Staubli VAL3: Robotscan.dtx

bool bSignal = true
bool bTxt1
bool bTxt2
bool bTxt3
bool btrig
public dio fout = {link=fOut0}
public frame FrmDraw = {x=1000, y=-100, fatherId=world[0]}
mdesc mNomSpeed
num l_nInit = 1500
num nNumTotal = 5031
num nNumrecord = 220
public num nTranC[6]
  [0] = 978.504226
  [1] = -109.919125
  [2] = 104.826018
  [3] = -0.09799
  [4] = 179.816018
  [5] = 56.0978696
num nTxtTotal = 11
num n_sTxt = 3
num ndelay = 16.304
public num nnnn = 2
num ntime = 2423.6
pointRx pfrmCad[1500]
  [0] = {x=-21.496, y=-9.92, z=104.826, rx=179.902, ry=0.184, rz=-123.901, fatherId=FrmDraw[0]}
  [1] = {x=-21.406, y=-9.571, z=104.833, rx=179.906, ry=0.177, rz=-124.352, fatherId=FrmDraw[0]}
  [2] = {x=-21.327, y=-9.235, z=104.84, rx=179.91, ry=0.172, rz=-124.769, fatherId=FrmDraw[0]}
  [3] = {x=-21.269, y=-8.967, z=104.845, rx=179.913, ry=0.168, rz=-125.087, fatherId=FrmDraw[0]}
  [4] = {x=-21.197, y=-8.609, z=104.852, rx=179.915, ry=0.164, rz=-125.501, fatherId=FrmDraw[0]}
  [5] = {x=-21.125, y=-8.284, z=104.858, rx=179.919, ry=0.159, rz=-125.914, fatherId=FrmDraw[0]}
  [6] = {x=-21.063, y=-8.029, z=104.863, rx=179.922, ry=0.154, rz=-126.277, fatherId=FrmDraw[0]}
  [7] = {x=-20.979, y=-7.711, z=104.871, rx=179.927, ry=0.146, rz=-126.778, fatherId=FrmDraw[0]}
  [8] = {x=-20.888, y=-7.402, z=104.879, rx=179.933, ry=0.136, rz=-127.324, fatherId=FrmDraw[0]}
  [9] = {x=-20.796, y=-7.121, z=104.886, rx=179.939, ry=0.125, rz=-127.88, fatherId=FrmDraw[0]}
  [10] = {x=-20.693, y=-6.864, z=104.895, rx=179.946, ry=0.112, rz=-128.514, fatherId=FrmDraw[0]}
  [11] = {x=-20.565, y=-6.611, z=104.905, rx=179.956, ry=0.094, rz=-129.312, fatherId=FrmDraw[0]}
  [12] = {x=-20.433, y=-6.398, z=104.914, rx=179.965, ry=0.076, rz=-130.171, fatherId=FrmDraw[0]}
  [13] = {x=-20.305, y=-6.222, z=104.923, rx=179.973, ry=0.059, rz=-131.051, fatherId=FrmDraw[0]}
  [14] = {x=-20.156, y=-6.043, z=104.933, rx=179.981, ry=0.042, rz=-132.148, fatherId=FrmDraw[0]}
  [15] = {x=-20.038, y=-5.901, z=104.94, rx=179.986, ry=0.032, rz=-133.098, fatherId=FrmDraw[0]}
  [16] = {x=-19.899, y=-5.734, z=104.948, rx=179.99, ry=0.023, rz=-134.309, fatherId=FrmDraw[0]}
  [17] = {x=-19.764, y=-5.576, z=104.955, rx=179.993, ry=0.017, rz=-135.558, fatherId=FrmDraw[0]}
  [18] = {x=-19.634, y=-5.431, z=104.961, rx=179.995, ry=0.013, rz=-136.824, fatherId=FrmDraw[0]}
  [19] = {x=-19.514, y=-5.306, z=104.967, rx=179.997, ry=0.008, rz=-138.02, fatherId=FrmDraw[0]}
  [20] = {x=-19.402, y=-5.193, z=104.973, rx=179.998, ry=0.005, rz=-139.156, fatherId=FrmDraw[0]}
  [21] = {x=-19.268, y=-5.059, z=104.979, rx=-180, rz=-140.558, fatherId=FrmDraw[0]}
  [22] = {x=-19.155, y=-4.95, z=104.985, rx=-179.999, ry=-0.004, rz=-141.768, fatherId=FrmDraw[0]}
  [23] = {x=-19.052, y=-4.852, z=104.99, rx=-179.997, ry=-0.008, rz=-142.893, fatherId=FrmDraw[0]}
  [24] = {x=-18.935, y=-4.744, z=104.995, rx=-179.996, ry=-0.013, rz=-144.181, fatherId=FrmDraw[0]}
  [25] = {x=-18.824, y=-4.636, z=105.001, rx=-179.995, ry=-0.017, rz=-145.451, fatherId=FrmDraw[0]}
  [26] = {x=-18.703, y=-4.509, z=105.006, rx=-179.994, ry=-0.021, rz=-146.89, fatherId=FrmDraw[0]}
  [27] = {x=-18.592, y=-4.383, z=105.011, rx=-179.993, ry=-0.023, rz=-148.26, fatherId=FrmDraw[0]}
  [28] = {x=-18.492, y=-4.26, z=105.016, rx=-179.993, ry=-0.024, rz=-149.572, fatherId=FrmDraw[0]}
  [29] = {x=-18.401, y=-4.137, z=105.02, rx=-179.994, ry=-0.023, rz=-150.833, fatherId=FrmDraw[0]}
  [30] = {x=-18.318, y=-4.016, z=105.023, rx=-179.995, ry=-0.022, rz=-152.05, fatherId=FrmDraw[0]}
  [31] = {x=-18.223, y=-3.864, z=105.027, rx=-179.996, ry=-0.017, rz=-153.555, fatherId=FrmDraw[0]}
  [32] = {x=-18.157, y=-3.747, z=105.029, rx=-179.997, ry=-0.012, rz=-154.683, fatherId=FrmDraw[0]}
  [33] = {x=-18.097, y=-3.632, z=105.031, rx=-179.999, ry=-0.006, rz=-155.782, fatherId=FrmDraw[0]}
  [34] = {x=-18.044, y=-3.519, z=105.032, rx=180, ry=0.001, rz=-156.854, fatherId=FrmDraw[0]}
  [35] = {x=-17.996, y=-3.408, z=105.033, rx=179.998, ry=0.01, rz=-157.905, fatherId=FrmDraw[0]}
  [36] = {x=-17.952, y=-3.3, z=105.034, rx=179.996, ry=0.019, rz=-158.942, fatherId=FrmDraw[0]}
  [37] = {x=-17.893, y=-3.145, z=105.035, rx=179.994, ry=0.034, rz=-160.472, fatherId=FrmDraw[0]}
  [38] = {x=-17.842, y=-2.998, z=105.035, rx=179.992, ry=0.05, rz=-161.989, fatherId=FrmDraw[0]}
  [39] = {x=-17.798, y=-2.858, z=105.034, rx=179.99, ry=0.068, rz=-163.483, fatherId=FrmDraw[0]}
  [40] = {x=-17.759, y=-2.726, z=105.033, rx=179.989, ry=0.087, rz=-164.962, fatherId=FrmDraw[0]}
  [41] = {x=-17.726, y=-2.601, z=105.032, rx=179.987, ry=0.106, rz=-166.428, fatherId=FrmDraw[0]}
  [42] = {x=-17.699, y=-2.483, z=105.03, rx=179.987, ry=0.127, rz=-167.883, fatherId=FrmDraw[0]}
  [43] = {x=-17.676, y=-2.372, z=105.028, rx=179.986, ry=0.148, rz=-169.329, fatherId=FrmDraw[0]}
  [44] = {x=-17.657, y=-2.266, z=105.026, rx=179.986, ry=0.17, rz=-170.767, fatherId=FrmDraw[0]}
  [45] = {x=-17.643, y=-2.167, z=105.023, rx=179.987, ry=0.193, rz=-172.197, fatherId=FrmDraw[0]}
  [46] = {x=-17.635, y=-2.07, z=105.02, rx=179.988, ry=0.217, rz=-173.604, fatherId=FrmDraw[0]}
  [47] = {x=-17.631, y=-1.974, z=105.016, rx=179.989, ry=0.242, rz=-174.986, fatherId=FrmDraw[0]}
  [48] = {x=-17.632, y=-1.879, z=105.012, rx=179.991, ry=0.268, rz=-176.347, fatherId=FrmDraw[0]}
  [49] = {x=-17.636, y=-1.787, z=105.008, rx=179.994, ry=0.293, rz=-177.689, fatherId=FrmDraw[0]}
  [50] = {x=-17.643, y=-1.696, z=105.004, rx=179.997, ry=0.319, rz=-179.015, fatherId=FrmDraw[0]}
  [51] = {x=-17.654, y=-1.579, z=104.998, rx=-179.998, ry=0.353, rz=179.235, fatherId=FrmDraw[0]}
  [52] = {x=-17.666, y=-1.469, z=104.993, rx=-179.992, ry=0.384, rz=177.491, fatherId=FrmDraw[0]}
  [53] = {x=-17.679, y=-1.366, z=104.987, rx=-179.985, ry=0.414, rz=175.749, fatherId=FrmDraw[0]}
  [54] = {x=-17.691, y=-1.271, z=104.982, rx=-179.977, ry=0.442, rz=174.006, fatherId=FrmDraw[0]}
  [55] = {x=-17.704, y=-1.183, z=104.977, rx=-179.968, ry=0.469, rz=172.258, fatherId=FrmDraw[0]}
  [56] = {x=-17.721, y=-1.092, z=104.972, rx=-179.959, ry=0.496, rz=170.546, fatherId=FrmDraw[0]}
  [57] = {x=-17.744, y=-0.993, z=104.966, rx=-179.949, ry=0.523, rz=168.902, fatherId=FrmDraw[0]}
  [58] = {x=-17.774, y=-0.886, z=104.96, rx=-179.939, ry=0.552, rz=167.322, fatherId=FrmDraw[0]}
  [59] = {x=-17.809, y=-0.77, z=104.954, rx=-179.928, ry=0.582, rz=165.802, fatherId=FrmDraw[0]}
  [60] = {x=-17.851, y=-0.646, z=104.947, rx=-179.916, ry=0.612, rz=164.339, fatherId=FrmDraw[0]}
  [61] = {x=-17.898, y=-0.515, z=104.94, rx=-179.903, ry=0.644, rz=162.93, fatherId=FrmDraw[0]}
  [62] = {x=-17.951, y=-0.376, z=104.932, rx=-179.89, ry=0.676, rz=161.572, fatherId=FrmDraw[0]}
  [63] = {x=-18.009, y=-0.231, z=104.925, rx=-179.877, ry=0.708, rz=160.261, fatherId=FrmDraw[0]}
  [64] = {x=-18.071, y=-0.079, z=104.917, rx=-179.863, ry=0.741, rz=158.995, fatherId=FrmDraw[0]}
  [65] = {x=-18.137, y=0.079, z=104.908, rx=-179.848, ry=0.775, rz=157.77, fatherId=FrmDraw[0]}
  [66] = {x=-18.207, y=0.239, z=104.9, rx=-179.833, ry=0.807, rz=156.562, fatherId=FrmDraw[0]}
  [67] = {x=-18.277, y=0.395, z=104.892, rx=-179.817, ry=0.839, rz=155.349, fatherId=FrmDraw[0]}
  [68] = {x=-18.35, y=0.548, z=104.885, rx=-179.8, ry=0.869, rz=154.132, fatherId=FrmDraw[0]}
  [69] = {x=-18.426, y=0.698, z=104.877, rx=-179.784, ry=0.898, rz=152.908, fatherId=FrmDraw[0]}
  [70] = {x=-18.504, y=0.844, z=104.869, rx=-179.766, ry=0.927, rz=151.676, fatherId=FrmDraw[0]}
  [71] = {x=-18.584, y=0.987, z=104.861, rx=-179.748, ry=0.955, rz=150.435, fatherId=FrmDraw[0]}
  [72] = {x=-18.668, y=1.126, z=104.854, rx=-179.729, ry=0.983, rz=149.184, fatherId=FrmDraw[0]}
  [73] = {x=-18.756, y=1.261, z=104.846, rx=-179.71, ry=1.01, rz=147.922, fatherId=FrmDraw[0]}
  [74] = {x=-18.847, y=1.391, z=104.838, rx=-179.689, ry=1.037, rz=146.647, fatherId=FrmDraw[0]}
  [75] = {x=-18.943, y=1.517, z=104.83, rx=-179.668, ry=1.064, rz=145.357, fatherId=FrmDraw[0]}
  [76] = {x=-19.043, y=1.64, z=104.821, rx=-179.646, ry=1.092, rz=144.066, fatherId=FrmDraw[0]}
  [77] = {x=-19.149, y=1.767, z=104.812, rx=-179.623, ry=1.121, rz=142.804, fatherId=FrmDraw[0]}
  [78] = {x=-19.258, y=1.9, z=104.803, rx=-179.599, ry=1.151, rz=141.57, fatherId=FrmDraw[0]}
  [79] = {x=-19.315, y=1.968, z=104.799, rx=-179.587, ry=1.166, rz=140.964, fatherId=FrmDraw[0]}
  [80] = {x=-19.401, y=2.072, z=104.792, rx=-179.568, ry=1.19, rz=140.069, fatherId=FrmDraw[0]}
  [81] = {x=-19.518, y=2.217, z=104.782, rx=-179.542, ry=1.221, rz=138.9, fatherId=FrmDraw[0]}
  [82] = {x=-19.638, y=2.368, z=104.772, rx=-179.516, ry=1.252, rz=137.76, fatherId=FrmDraw[0]}
  [83] = {x=-19.759, y=2.525, z=104.763, rx=-179.49, ry=1.282, rz=136.648, fatherId=FrmDraw[0]}
  [84] = {x=-19.88, y=2.688, z=104.754, rx=-179.464, ry=1.312, rz=135.564, fatherId=FrmDraw[0]}
  [85] = {x=-20.001, y=2.86, z=104.745, rx=-179.438, ry=1.34, rz=134.508, fatherId=FrmDraw[0]}
  [86] = {x=-20.122, y=3.039, z=104.736, rx=-179.412, ry=1.367, rz=133.478, fatherId=FrmDraw[0]}
  [87] = {x=-20.24, y=3.225, z=104.728, rx=-179.387, ry=1.391, rz=132.471, fatherId=FrmDraw[0]}
  [88] = {x=-20.358, y=3.418, z=104.721, rx=-179.363, ry=1.413, rz=131.482, fatherId=FrmDraw[0]}
  [89] = {x=-20.475, y=3.617, z=104.714, rx=-179.339, ry=1.434, rz=130.511, fatherId=FrmDraw[0]}
  [90] = {x=-20.592, y=3.823, z=104.707, rx=-179.316, ry=1.453, rz=129.559, fatherId=FrmDraw[0]}
  [91] = {x=-20.71, y=4.035, z=104.701, rx=-179.293, ry=1.471, rz=128.624, fatherId=FrmDraw[0]}
  [92] = {x=-20.823, y=4.242, z=104.695, rx=-179.271, ry=1.487, rz=127.752, fatherId=FrmDraw[0]}
  [93] = {x=-20.943, y=4.465, z=104.689, rx=-179.248, ry=1.504, rz=126.851, fatherId=FrmDraw[0]}
  [94] = {x=-21.066, y=4.694, z=104.683, rx=-179.224, ry=1.521, rz=125.967, fatherId=FrmDraw[0]}
  [95] = {x=-21.192, y=4.928, z=104.677, rx=-179.201, ry=1.538, rz=125.099, fatherId=FrmDraw[0]}
  [96] = {x=-21.321, y=5.168, z=104.67, rx=-179.177, ry=1.556, rz=124.249, fatherId=FrmDraw[0]}
  [97] = {x=-21.453, y=5.415, z=104.664, rx=-179.153, ry=1.575, rz=123.427, fatherId=FrmDraw[0]}
  [98] = {x=-21.587, y=5.671, z=104.658, rx=-179.128, ry=1.594, rz=122.636, fatherId=FrmDraw[0]}
  [99] = {x=-21.722, y=5.937, z=104.652, rx=-179.103, ry=1.615, rz=121.878, fatherId=FrmDraw[0]}
  [100] = {x=-21.857, y=6.213, z=104.646, rx=-179.078, ry=1.635, rz=121.155, fatherId=FrmDraw[0]}
  [101] = {x=-21.99, y=6.5, z=104.64, rx=-179.053, ry=1.655, rz=120.468, fatherId=FrmDraw[0]}
  [102] = {x=-22.118, y=6.791, z=104.635, rx=-179.03, ry=1.674, rz=119.831, fatherId=FrmDraw[0]}
  [103] = {x=-22.226, y=7.051, z=104.631, rx=-179.011, ry=1.69, rz=119.312, fatherId=FrmDraw[0]}
  [104] = {x=-22.313, y=7.274, z=104.628, rx=-178.995, ry=1.702, rz=118.9, fatherId=FrmDraw[0]}
  [105] = {x=-22.431, y=7.598, z=104.624, rx=-178.975, ry=1.718, rz=118.352, fatherId=FrmDraw[0]}
  [106] = {x=-22.528, y=7.887, z=104.622, rx=-178.958, ry=1.731, rz=117.91, fatherId=FrmDraw[0]}
  [107] = {x=-22.602, y=8.124, z=104.62, rx=-178.946, ry=1.74, rz=117.572, fatherId=FrmDraw[0]}
  [108] = {x=-22.692, y=8.429, z=104.618, rx=-178.931, ry=1.75, rz=117.171, fatherId=FrmDraw[0]}
  [109] = {x=-22.762, y=8.68, z=104.617, rx=-178.92, ry=1.757, rz=116.866, fatherId=FrmDraw[0]}
  [110] = {x=-22.845, y=9.001, z=104.617, rx=-178.908, ry=1.765, rz=116.506, fatherId=FrmDraw[0]}
  [111] = {x=-22.909, y=9.265, z=104.616, rx=-178.898, ry=1.772, rz=116.235, fatherId=FrmDraw[0]}
  [112] = {x=-22.985, y=9.602, z=104.616, rx=-178.887, ry=1.779, rz=115.918, fatherId=FrmDraw[0]}
  [113] = {x=-23.044, y=9.878, z=104.616, rx=-178.878, ry=1.784, rz=115.682, fatherId=FrmDraw[0]}
  [114] = {x=-23.114, y=10.232, z=104.616, rx=-178.868, ry=1.791, rz=115.409, fatherId=FrmDraw[0]}
  [115] = {x=-23.168, y=10.52, z=104.617, rx=-178.86, ry=1.797, rz=115.209, fatherId=FrmDraw[0]}
  [116] = {x=-23.231, y=10.889, z=104.617, rx=-178.85, ry=1.804, rz=114.981, fatherId=FrmDraw[0]}
  [117] = {x=-23.28, y=11.188, z=104.618, rx=-178.843, ry=1.809, rz=114.813, fatherId=FrmDraw[0]}
  [118] = {x=-23.341, y=11.564, z=104.619, rx=-178.834, ry=1.816, rz=114.603, fatherId=FrmDraw[0]}
  [119] = {x=-23.391, y=11.865, z=104.62, rx=-178.827, ry=1.821, rz=114.433, fatherId=FrmDraw[0]}
  [120] = {x=-23.455, y=12.243, z=104.621, rx=-178.819, ry=1.827, rz=114.218, fatherId=FrmDraw[0]}
  [121] = {x=-23.507, y=12.545, z=104.623, rx=-178.812, ry=1.831, rz=114.045, fatherId=FrmDraw[0]}
  [122] = {x=-23.573, y=12.924, z=104.624, rx=-178.804, ry=1.836, rz=113.827, fatherId=FrmDraw[0]}
  [123] = {x=-23.626, y=13.227, z=104.625, rx=-178.797, ry=1.84, rz=113.651, fatherId=FrmDraw[0]}
  [124] = {x=-23.695, y=13.607, z=104.627, rx=-178.789, ry=1.844, rz=113.428, fatherId=FrmDraw[0]}
  [125] = {x=-23.751, y=13.912, z=104.628, rx=-178.783, ry=1.847, rz=113.248, fatherId=FrmDraw[0]}
  [126] = {x=-23.823, y=14.293, z=104.63, rx=-178.775, ry=1.851, rz=113.022, fatherId=FrmDraw[0]}
  [127] = {x=-23.882, y=14.598, z=104.632, rx=-178.769, ry=1.854, rz=112.839, fatherId=FrmDraw[0]}
  [128] = {x=-23.957, y=14.981, z=104.634, rx=-178.761, ry=1.858, rz=112.607, fatherId=FrmDraw[0]}
  [129] = {x=-24.019, y=15.287, z=104.635, rx=-178.755, ry=1.861, rz=112.421, fatherId=FrmDraw[0]}
  [130] = {x=-24.098, y=15.67, z=104.637, rx=-178.747, ry=1.864, rz=112.186, fatherId=FrmDraw[0]}
  [131] = {x=-24.163, y=15.977, z=104.639, rx=-178.741, ry=1.867, rz=111.995, fatherId=FrmDraw[0]}
  [132] = {x=-24.246, y=16.361, z=104.641, rx=-178.733, ry=1.87, rz=111.755, fatherId=FrmDraw[0]}
  [133] = {x=-24.315, y=16.668, z=104.642, rx=-178.726, ry=1.873, rz=111.562, fatherId=FrmDraw[0]}
  [134] = {x=-24.403, y=17.053, z=104.645, rx=-178.718, ry=1.877, rz=111.317, fatherId=FrmDraw[0]}
  [135] = {x=-24.476, y=17.36, z=104.646, rx=-178.711, ry=1.88, rz=111.12, fatherId=FrmDraw[0]}
  [136] = {x=-24.57, y=17.745, z=104.648, rx=-178.702, ry=1.883, rz=110.87, fatherId=FrmDraw[0]}
  [137] = {x=-24.647, y=18.053, z=104.65, rx=-178.695, ry=1.887, rz=110.669, fatherId=FrmDraw[0]}
  [138] = {x=-24.746, y=18.438, z=104.652, rx=-178.686, ry=1.891, rz=110.415, fatherId=FrmDraw[0]}
  [139] = {x=-24.827, y=18.746, z=104.654, rx=-178.678, ry=1.895, rz=110.213, fatherId=FrmDraw[0]}
  [140] = {x=-24.929, y=19.134, z=104.656, rx=-178.669, ry=1.9, rz=109.963, fatherId=FrmDraw[0]}
  [141] = {x=-25.011, y=19.446, z=104.657, rx=-178.661, ry=1.904, rz=109.767, fatherId=FrmDraw[0]}
  [142] = {x=-25.114, y=19.839, z=104.66, rx=-178.651, ry=1.909, rz=109.526, fatherId=FrmDraw[0]}
  [143] = {x=-25.196, y=20.155, z=104.662, rx=-178.643, ry=1.914, rz=109.336, fatherId=FrmDraw[0]}
  [144] = {x=-25.298, y=20.553, z=104.664, rx=-178.634, ry=1.918, rz=109.102, fatherId=FrmDraw[0]}
  [145] = {x=-25.378, y=20.875, z=104.667, rx=-178.627, ry=1.922, rz=108.919, fatherId=FrmDraw[0]}
  [146] = {x=-25.478, y=21.279, z=104.67, rx=-178.619, ry=1.925, rz=108.693, fatherId=FrmDraw[0]}
  [147] = {x=-25.556, y=21.606, z=104.672, rx=-178.613, ry=1.928, rz=108.516, fatherId=FrmDraw[0]}
  [148] = {x=-25.651, y=22.019, z=104.675, rx=-178.606, ry=1.929, rz=108.299, fatherId=FrmDraw[0]}
  [149] = {x=-25.727, y=22.351, z=104.678, rx=-178.601, ry=1.93, rz=108.126, fatherId=FrmDraw[0]}
  [150] = {x=-25.823, y=22.767, z=104.682, rx=-178.596, ry=1.929, rz=107.903, fatherId=FrmDraw[0]}
  [151] = {x=-25.901, y=23.101, z=104.684, rx=-178.592, ry=1.928, rz=107.72, fatherId=FrmDraw[0]}
  [152] = {x=-26.003, y=23.518, z=104.688, rx=-178.588, ry=1.925, rz=107.485, fatherId=FrmDraw[0]}
  [153] = {x=-26.087, y=23.851, z=104.691, rx=-178.585, ry=1.923, rz=107.292, fatherId=FrmDraw[0]}
  [154] = {x=-26.197, y=24.266, z=104.694, rx=-178.58, ry=1.92, rz=107.045, fatherId=FrmDraw[0]}
  [155] = {x=-26.31, y=24.666, z=104.697, rx=-178.575, ry=1.918, rz=106.799, fatherId=FrmDraw[0]}
  [156] = {x=-26.411, y=25.01, z=104.7, rx=-178.571, ry=1.917, rz=106.581, fatherId=FrmDraw[0]}
  [157] = {x=-26.536, y=25.406, z=104.703, rx=-178.564, ry=1.916, rz=106.322, fatherId=FrmDraw[0]}
  [158] = {x=-26.745, y=25.675, z=104.703, rx=-178.557, ry=1.911, rz=105.881, fatherId=FrmDraw[0]}
  [159] = {x=-26.744, y=25.675, z=105.202, rx=-178.556, ry=1.913, rz=105.887, fatherId=FrmDraw[0]}
  [160] = {x=-26.743, y=25.675, z=105.702, rx=-178.555, ry=1.914, rz=105.893, fatherId=FrmDraw[0]}
  [161] = {x=-26.743, y=25.675, z=106.101, rx=-178.554, ry=1.915, rz=105.898, fatherId=FrmDraw[0]}
  [162] = {x=-26.742, y=25.675, z=106.501, rx=-178.554, ry=1.916, rz=105.903, fatherId=FrmDraw[0]}
  [163] = {x=-26.742, y=25.675, z=106.74, rx=-178.553, ry=1.917, rz=105.906, fatherId=FrmDraw[0]}
  [164] = {x=-26.742, y=25.675, z=107.1, rx=-178.553, ry=1.918, rz=105.91, fatherId=FrmDraw[0]}
  [165] = {x=-26.741, y=25.674, z=107.578, rx=-178.552, ry=1.919, rz=105.916, fatherId=FrmDraw[0]}
  [166] = {x=-26.741, y=25.674, z=108.029, rx=-178.551, ry=1.92, rz=105.921, fatherId=FrmDraw[0]}
  [167] = {x=-26.74, y=25.674, z=108.403, rx=-178.55, ry=1.921, rz=105.926, fatherId=FrmDraw[0]}
  [168] = {x=-26.74, y=25.674, z=108.777, rx=-178.55, ry=1.922, rz=105.93, fatherId=FrmDraw[0]}
  [169] = {x=-26.577, y=25.37, z=108.776, rx=-178.554, ry=1.929, rz=106.286, fatherId=FrmDraw[0]}
  [170] = {x=-26.456, y=24.972, z=108.772, rx=-178.558, ry=1.932, rz=106.549, fatherId=FrmDraw[0]}
  [171] = {x=-26.355, y=24.627, z=108.77, rx=-178.562, ry=1.935, rz=106.769, fatherId=FrmDraw[0]}
  [172] = {x=-26.243, y=24.227, z=108.766, rx=-178.566, ry=1.938, rz=107.016, fatherId=FrmDraw[0]}
  [173] = {x=-26.132, y=23.812, z=108.763, rx=-178.572, ry=1.94, rz=107.263, fatherId=FrmDraw[0]}
  [174] = {x=-26.046, y=23.48, z=108.76, rx=-178.576, ry=1.941, rz=107.454, fatherId=FrmDraw[0]}
  [175] = {x=-25.943, y=23.065, z=108.757, rx=-178.581, ry=1.941, rz=107.685, fatherId=FrmDraw[0]}
  [176] = {x=-25.863, y=22.732, z=108.754, rx=-178.586, ry=1.941, rz=107.863, fatherId=FrmDraw[0]}
  [177] = {x=-25.766, y=22.316, z=108.75, rx=-178.592, ry=1.94, rz=108.078, fatherId=FrmDraw[0]}
  [178] = {x=-25.691, y=21.983, z=108.748, rx=-178.598, ry=1.938, rz=108.244, fatherId=FrmDraw[0]}
  [179] = {x=-25.597, y=21.568, z=108.744, rx=-178.605, ry=1.936, rz=108.453, fatherId=FrmDraw[0]}
  [180] = {x=-25.521, y=21.24, z=108.742, rx=-178.611, ry=1.934, rz=108.625, fatherId=FrmDraw[0]}
  [181] = {x=-25.424, y=20.833, z=108.739, rx=-178.619, ry=1.93, rz=108.844, fatherId=FrmDraw[0]}
  [182] = {x=-25.346, y=20.51, z=108.736, rx=-178.626, ry=1.927, rz=109.024, fatherId=FrmDraw[0]}
  [183] = {x=-25.247, y=20.109, z=108.733, rx=-178.634, ry=1.924, rz=109.254, fatherId=FrmDraw[0]}
  [184] = {x=-25.167, y=19.791, z=108.731, rx=-178.641, ry=1.921, rz=109.442, fatherId=FrmDraw[0]}
  [185] = {x=-25.067, y=19.396, z=108.729, rx=-178.65, ry=1.917, rz=109.683, fatherId=FrmDraw[0]}
  [186] = {x=-24.987, y=19.083, z=108.727, rx=-178.657, ry=1.914, rz=109.879, fatherId=FrmDraw[0]}
  [187] = {x=-24.886, y=18.694, z=108.724, rx=-178.666, ry=1.91, rz=110.129, fatherId=FrmDraw[0]}
  [188] = {x=-24.806, y=18.384, z=108.723, rx=-178.673, ry=1.907, rz=110.333, fatherId=FrmDraw[0]}
  [189] = {x=-24.707, y=17.999, z=108.72, rx=-178.681, ry=1.904, rz=110.589, fatherId=FrmDraw[0]}
  [190] = {x=-24.63, y=17.691, z=108.719, rx=-178.688, ry=1.901, rz=110.792, fatherId=FrmDraw[0]}
  [191] = {x=-24.537, y=17.306, z=108.716, rx=-178.697, ry=1.898, rz=111.043, fatherId=FrmDraw[0]}
  [192] = {x=-24.464, y=16.999, z=108.715, rx=-178.703, ry=1.895, rz=111.241, fatherId=FrmDraw[0]}
  [193] = {x=-24.375, y=16.615, z=108.712, rx=-178.712, ry=1.892, rz=111.486, fatherId=FrmDraw[0]}
  [194] = {x=-24.305, y=16.308, z=108.711, rx=-178.718, ry=1.889, rz=111.681, fatherId=FrmDraw[0]}
  [195] = {x=-24.221, y=15.924, z=108.709, rx=-178.726, ry=1.885, rz=111.921, fatherId=FrmDraw[0]}
  [196] = {x=-24.155, y=15.618, z=108.707, rx=-178.733, ry=1.882, rz=112.111, fatherId=FrmDraw[0]}
  [197] = {x=-24.074, y=15.236, z=108.705, rx=-178.741, ry=1.878, rz=112.345, fatherId=FrmDraw[0]}
  [198] = {x=-24.011, y=14.93, z=108.704, rx=-178.748, ry=1.875, rz=112.531, fatherId=FrmDraw[0]}
  [199] = {x=-23.935, y=14.548, z=108.702, rx=-178.756, ry=1.871, rz=112.761, fatherId=FrmDraw[0]}
  [200] = {x=-23.875, y=14.243, z=108.7, rx=-178.763, ry=1.867, rz=112.943, fatherId=FrmDraw[0]}
  [201] = {x=-23.802, y=13.863, z=108.698, rx=-178.771, ry=1.862, rz=113.169, fatherId=FrmDraw[0]}
  [202] = {x=-23.744, y=13.559, z=108.697, rx=-178.778, ry=1.859, rz=113.347, fatherId=FrmDraw[0]}
  [203] = {x=-23.674, y=13.179, z=108.696, rx=-178.786, ry=1.853, rz=113.567, fatherId=FrmDraw[0]}
  [204] = {x=-23.62, y=12.876, z=108.694, rx=-178.793, ry=1.849, rz=113.741, fatherId=FrmDraw[0]}
  [205] = {x=-23.552, y=12.497, z=108.693, rx=-178.802, ry=1.843, rz=113.957, fatherId=FrmDraw[0]}
  [206] = {x=-23.5, y=12.195, z=108.692, rx=-178.809, ry=1.839, rz=114.128, fatherId=FrmDraw[0]}
  [207] = {x=-23.435, y=11.818, z=108.69, rx=-178.818, ry=1.832, rz=114.339, fatherId=FrmDraw[0]}
  [208] = {x=-23.385, y=11.516, z=108.689, rx=-178.825, ry=1.827, rz=114.506, fatherId=FrmDraw[0]}
  [209] = {x=-23.323, y=11.14, z=108.688, rx=-178.834, ry=1.82, rz=114.713, fatherId=FrmDraw[0]}
  [210] = {x=-23.274, y=10.84, z=108.688, rx=-178.841, ry=1.814, rz=114.879, fatherId=FrmDraw[0]}
  [211] = {x=-23.21, y=10.471, z=108.687, rx=-178.851, ry=1.807, rz=115.105, fatherId=FrmDraw[0]}
  [212] = {x=-23.156, y=10.182, z=108.686, rx=-178.859, ry=1.802, rz=115.303, fatherId=FrmDraw[0]}
  [213] = {x=-23.086, y=9.828, z=108.686, rx=-178.869, ry=1.795, rz=115.571, fatherId=FrmDraw[0]}
  [214] = {x=-23.028, y=9.55, z=108.686, rx=-178.878, ry=1.789, rz=115.802, fatherId=FrmDraw[0]}
  [215] = {x=-22.952, y=9.21, z=108.686, rx=-178.889, ry=1.782, rz=116.11, fatherId=FrmDraw[0]}
  [216] = {x=-22.889, y=8.945, z=108.686, rx=-178.899, ry=1.775, rz=116.373, fatherId=FrmDraw[0]}
  [217] = {x=-22.806, y=8.621, z=108.687, rx=-178.912, ry=1.766, rz=116.721, fatherId=FrmDraw[0]}
  [218] = {x=-22.737, y=8.368, z=108.688, rx=-178.923, ry=1.759, rz=117.016, fatherId=FrmDraw[0]}
  [219] = {x=-22.656, y=8.09, z=108.69, rx=-178.936, ry=1.749, rz=117.363, fatherId=FrmDraw[0]}
  [220] = {x=-22.572, y=7.82, z=108.692, rx=-178.95, ry=1.738, rz=117.728, fatherId=FrmDraw[0]}
  [221] = {x=-22.475, y=7.528, z=108.695, rx=-178.967, ry=1.724, rz=118.152, fatherId=FrmDraw[0]}
  [222] = {x=-22.355, y=7.201, z=108.699, rx=-178.988, ry=1.706, rz=118.682, fatherId=FrmDraw[0]}
  [223] = {x=-22.267, y=6.976, z=108.702, rx=-179.004, ry=1.693, rz=119.085, fatherId=FrmDraw[0]}
  [224] = {x=-22.157, y=6.715, z=108.706, rx=-179.024, ry=1.676, rz=119.593, fatherId=FrmDraw[0]}
  [225] = {x=-22.026, y=6.423, z=108.711, rx=-179.048, ry=1.656, rz=120.221, fatherId=FrmDraw[0]}
  [226] = {x=-21.89, y=6.136, z=108.717, rx=-179.074, ry=1.634, rz=120.903, fatherId=FrmDraw[0]}
  [227] = {x=-21.752, y=5.86, z=108.724, rx=-179.099, ry=1.613, rz=121.625, fatherId=FrmDraw[0]}
  [228] = {x=-21.615, y=5.596, z=108.73, rx=-179.124, ry=1.592, rz=122.385, fatherId=FrmDraw[0]}
  [229] = {x=-21.478, y=5.341, z=108.736, rx=-179.15, ry=1.572, rz=123.182, fatherId=FrmDraw[0]}
  [230] = {x=-21.344, y=5.097, z=108.742, rx=-179.174, ry=1.553, rz=124.013, fatherId=FrmDraw[0]}
  [231] = {x=-21.213, y=4.859, z=108.748, rx=-179.198, ry=1.536, rz=124.871, fatherId=FrmDraw[0]}
  [232] = {x=-21.087, y=4.625, z=108.754, rx=-179.221, ry=1.519, rz=125.743, fatherId=FrmDraw[0]}
  [233] = {x=-20.964, y=4.397, z=108.76, rx=-179.244, ry=1.503, rz=126.629, fatherId=FrmDraw[0]}
  [234] = {x=-20.843, y=4.173, z=108.766, rx=-179.267, ry=1.486, rz=127.529, fatherId=FrmDraw[0]}
  [235] = {x=-20.73, y=3.965, z=108.772, rx=-179.289, ry=1.47, rz=128.397, fatherId=FrmDraw[0]}
  [236] = {x=-20.612, y=3.751, z=108.778, rx=-179.312, ry=1.452, rz=129.324, fatherId=FrmDraw[0]}
  [237] = {x=-20.495, y=3.543, z=108.785, rx=-179.336, ry=1.433, rz=130.267, fatherId=FrmDraw[0]}
  [238] = {x=-20.377, y=3.341, z=108.792, rx=-179.36, ry=1.413, rz=131.224, fatherId=FrmDraw[0]}
  [239] = {x=-20.259, y=3.144, z=108.8, rx=-179.384, ry=1.39, rz=132.196, fatherId=FrmDraw[0]}
  [240] = {x=-20.139, y=2.954, z=108.808, rx=-179.409, ry=1.365, rz=133.183, fatherId=FrmDraw[0]}
  [241] = {x=-20.017, y=2.772, z=108.817, rx=-179.435, ry=1.337, rz=134.197, fatherId=FrmDraw[0]}
  [242] = {x=-19.894, y=2.599, z=108.826, rx=-179.461, ry=1.309, rz=135.242, fatherId=FrmDraw[0]}
  [243] = {x=-19.772, y=2.434, z=108.835, rx=-179.487, ry=1.279, rz=136.319, fatherId=FrmDraw[0]}
  [244] = {x=-19.65, y=2.276, z=108.845, rx=-179.514, ry=1.248, rz=137.427, fatherId=FrmDraw[0]}
  [245] = {x=-19.53, y=2.126, z=108.854, rx=-179.54, ry=1.218, rz=138.567, fatherId=FrmDraw[0]}
  [246] = {x=-19.412, y=1.983, z=108.864, rx=-179.565, ry=1.187, rz=139.739, fatherId=FrmDraw[0]}
  [247] = {x=-19.297, y=1.846, z=108.873, rx=-179.59, ry=1.156, rz=140.944, fatherId=FrmDraw[0]}
  [248] = {x=-19.186, y=1.714, z=108.882, rx=-179.614, ry=1.127, rz=142.182, fatherId=FrmDraw[0]}
  [249] = {x=-19.08, y=1.589, z=108.891, rx=-179.637, ry=1.099, rz=143.452, fatherId=FrmDraw[0]}
  [250] = {x=-18.979, y=1.468, z=108.899, rx=-179.659, ry=1.072, rz=144.753, fatherId=FrmDraw[0]}
  [251] = {x=-18.883, y=1.345, z=108.907, rx=-179.681, ry=1.046, rz=146.05, fatherId=FrmDraw[0]}
  [252] = {x=-18.791, y=1.217, z=108.915, rx=-179.701, ry=1.019, rz=147.331, fatherId=FrmDraw[0]}
  [253] = {x=-18.703, y=1.084, z=108.923, rx=-179.721, ry=0.992, rz=148.598, fatherId=FrmDraw[0]}
  [254] = {x=-18.618, y=0.946, z=108.93, rx=-179.74, ry=0.965, rz=149.852, fatherId=FrmDraw[0]}
  [255] = {x=-18.536, y=0.804, z=108.938, rx=-179.758, ry=0.938, rz=151.094, fatherId=FrmDraw[0]}
  [256] = {x=-18.457, y=0.659, z=108.946, rx=-179.776, ry=0.909, rz=152.325, fatherId=FrmDraw[0]}
  [257] = {x=-18.382, y=0.509, z=108.953, rx=-179.793, ry=0.881, rz=153.546, fatherId=FrmDraw[0]}
  [258] = {x=-18.308, y=0.356, z=108.961, rx=-179.809, ry=0.851, rz=154.76, fatherId=FrmDraw[0]}
  [259] = {x=-18.238, y=0.199, z=108.969, rx=-179.825, ry=0.821, rz=155.966, fatherId=FrmDraw[0]}
  [260] = {x=-18.169, y=0.039, z=108.977, rx=-179.841, ry=0.79, rz=157.167, fatherId=FrmDraw[0]}
  [261] = {x=-18.104, y=-0.119, z=108.984, rx=-179.855, ry=0.758, rz=158.386, fatherId=FrmDraw[0]}
  [262] = {x=-18.044, y=-0.27, z=108.992, rx=-179.869, ry=0.727, rz=159.648, fatherId=FrmDraw[0]}
  [263] = {x=-17.988, y=-0.416, z=108.999, rx=-179.883, ry=0.697, rz=160.955, fatherId=FrmDraw[0]}
  [264] = {x=-17.938, y=-0.554, z=109.006, rx=-179.896, ry=0.667, rz=162.309, fatherId=FrmDraw[0]}
  [265] = {x=-17.893, y=-0.685, z=109.013, rx=-179.909, ry=0.638, rz=163.713, fatherId=FrmDraw[0]}
  [266] = {x=-17.854, y=-0.808, z=109.02, rx=-179.921, ry=0.609, rz=165.171, fatherId=FrmDraw[0]}
  [267] = {x=-17.819, y=-0.923, z=109.026, rx=-179.932, ry=0.581, rz=166.685, fatherId=FrmDraw[0]}
  [268] = {x=-17.79, y=-1.03, z=109.032, rx=-179.943, ry=0.553, rz=168.259, fatherId=FrmDraw[0]}
  [269] = {x=-17.766, y=-1.128, z=109.037, rx=-179.954, ry=0.526, rz=169.896, fatherId=FrmDraw[0]}
  [270] = {x=-17.747, y=-1.217, z=109.043, rx=-179.963, ry=0.499, rz=171.6, fatherId=FrmDraw[0]}
  [271] = {x=-17.729, y=-1.306, z=109.048, rx=-179.973, ry=0.47, rz=173.332, fatherId=FrmDraw[0]}
  [272] = {x=-17.71, y=-1.401, z=109.054, rx=-179.981, ry=0.44, rz=175.061, fatherId=FrmDraw[0]}
  [273] = {x=-17.691, y=-1.503, z=109.06, rx=-179.989, ry=0.407, rz=176.789, fatherId=FrmDraw[0]}
  [274] = {x=-17.672, y=-1.612, z=109.066, rx=-179.995, ry=0.373, rz=178.52, fatherId=FrmDraw[0]}
  [275] = {x=-17.656, y=-1.728, z=109.072, rx=179.999, ry=0.338, rz=-179.741, fatherId=FrmDraw[0]}
  [276] = {x=-17.643, y=-1.847, z=109.078, rx=179.995, ry=0.302, rz=-177.976, fatherId=FrmDraw[0]}
  [277] = {x=-17.638, y=-1.937, z=109.083, rx=179.992, ry=0.276, rz=-176.631, fatherId=FrmDraw[0]}
  [278] = {x=-17.638, y=-2.029, z=109.086, rx=179.99, ry=0.251, rz=-175.263, fatherId=FrmDraw[0]}
  [279] = {x=-17.642, y=-2.121, z=109.09, rx=179.988, ry=0.226, rz=-173.871, fatherId=FrmDraw[0]}
  [280] = {x=-17.653, y=-2.214, z=109.093, rx=179.987, ry=0.203, rz=-172.45, fatherId=FrmDraw[0]}
  [281] = {x=-17.668, y=-2.309, z=109.096, rx=179.986, ry=0.181, rz=-171.012, fatherId=FrmDraw[0]}
  [282] = {x=-17.688, y=-2.411, z=109.098, rx=179.985, ry=0.16, rz=-169.567, fatherId=FrmDraw[0]}
  [283] = {x=-17.712, y=-2.519, z=109.1, rx=179.985, ry=0.139, rz=-168.114, fatherId=FrmDraw[0]}
  [284] = {x=-17.741, y=-2.634, z=109.101, rx=179.986, ry=0.12, rz=-166.653, fatherId=FrmDraw[0]}
  [285] = {x=-17.775, y=-2.756, z=109.103, rx=179.987, ry=0.101, rz=-165.18, fatherId=FrmDraw[0]}
  [286] = {x=-17.814, y=-2.884, z=109.103, rx=179.988, ry=0.083, rz=-163.694, fatherId=FrmDraw[0]}
  [287] = {x=-17.86, y=-3.02, z=109.104, rx=179.99, ry=0.066, rz=-162.192, fatherId=FrmDraw[0]}
  [288] = {x=-17.911, y=-3.162, z=109.104, rx=179.992, ry=0.05, rz=-160.677, fatherId=FrmDraw[0]}
  [289] = {x=-17.971, y=-3.313, z=109.103, rx=179.994, ry=0.035, rz=-159.128, fatherId=FrmDraw[0]}
  [290] = {x=-18.037, y=-3.468, z=109.102, rx=179.996, ry=0.022, rz=-157.586, fatherId=FrmDraw[0]}
  [291] = {x=-18.088, y=-3.576, z=109.101, rx=179.997, ry=0.014, rz=-156.527, fatherId=FrmDraw[0]}
  [292] = {x=-18.144, y=-3.684, z=109.099, rx=179.998, ry=0.007, rz=-155.445, fatherId=FrmDraw[0]}
  [293] = {x=-18.206, y=-3.795, z=109.097, rx=180, ry=0.002, rz=-154.337, fatherId=FrmDraw[0]}
  [294] = {x=-18.274, y=-3.907, z=109.095, rx=-179.999, ry=-0.003, rz=-153.2, fatherId=FrmDraw[0]}
  [295] = {x=-18.349, y=-4.02, z=109.092, rx=-179.999, ry=-0.006, rz=-152.031, fatherId=FrmDraw[0]}
  [296] = {x=-18.431, y=-4.135, z=109.089, rx=-179.998, ry=-0.008, rz=-150.826, fatherId=FrmDraw[0]}
  [297] = {x=-18.52, y=-4.251, z=109.085, rx=-179.998, ry=-0.008, rz=-149.58, fatherId=FrmDraw[0]}
  [298] = {x=-18.619, y=-4.369, z=109.081, rx=-179.998, ry=-0.008, rz=-148.288, fatherId=FrmDraw[0]}
  [299] = {x=-18.726, y=-4.488, z=109.076, rx=-179.998, ry=-0.006, rz=-146.943, fatherId=FrmDraw[0]}
  [300] = {x=-18.844, y=-4.609, z=109.07, rx=-179.999, ry=-0.003, rz=-145.536, fatherId=FrmDraw[0]}
  [301] = {x=-18.974, y=-4.731, z=109.064, rx=179.999, ry=0.002, rz=-144.053, fatherId=FrmDraw[0]}
  [302] = {x=-19.07, y=-4.82, z=109.06, rx=179.998, ry=0.006, rz=-142.989, fatherId=FrmDraw[0]}
  [303] = {x=-19.19, y=-4.932, z=109.054, rx=179.996, ry=0.011, rz=-141.688, fatherId=FrmDraw[0]}
  [304] = {x=-19.313, y=-5.049, z=109.048, rx=179.994, ry=0.016, rz=-140.393, fatherId=FrmDraw[0]}
  [305] = {x=-19.431, y=-5.162, z=109.042, rx=179.992, ry=0.021, rz=-139.184, fatherId=FrmDraw[0]}
  [306] = {x=-19.564, y=-5.291, z=109.035, rx=179.989, ry=0.028, rz=-137.86, fatherId=FrmDraw[0]}
  [307] = {x=-19.689, y=-5.411, z=109.029, rx=179.986, ry=0.034, rz=-136.673, fatherId=FrmDraw[0]}
  [308] = {x=-19.819, y=-5.541, z=109.021, rx=179.983, ry=0.043, rz=-135.477, fatherId=FrmDraw[0]}
  [309] = {x=-19.965, y=-5.687, z=109.013, rx=179.977, ry=0.054, rz=-134.218, fatherId=FrmDraw[0]}
  [310] = {x=-20.089, y=-5.808, z=109.006, rx=179.971, ry=0.066, rz=-133.222, fatherId=FrmDraw[0]}
  [311] = {x=-20.24, y=-5.95, z=108.996, rx=179.963, ry=0.084, rz=-132.095, fatherId=FrmDraw[0]}
  [312] = {x=-20.396, y=-6.104, z=108.986, rx=179.952, ry=0.106, rz=-131.024, fatherId=FrmDraw[0]}
  [313] = {x=-20.534, y=-6.268, z=108.976, rx=179.941, ry=0.127, rz=-130.13, fatherId=FrmDraw[0]}
  [314] = {x=-20.675, y=-6.476, z=108.966, rx=179.929, ry=0.149, rz=-129.253, fatherId=FrmDraw[0]}
  [315] = {x=-20.81, y=-6.725, z=108.955, rx=179.918, ry=0.171, rz=-128.457, fatherId=FrmDraw[0]}
  [316] = {x=-20.918, y=-6.986, z=108.946, rx=179.908, ry=0.188, rz=-127.832, fatherId=FrmDraw[0]}
  [317] = {x=-21.001, y=-7.219, z=108.939, rx=179.901, ry=0.2, rz=-127.367, fatherId=FrmDraw[0]}
  [318] = {x=-21.104, y=-7.533, z=108.93, rx=179.892, ry=0.215, rz=-126.805, fatherId=FrmDraw[0]}
  [319] = {x=-21.199, y=-7.86, z=108.921, rx=179.885, ry=0.228, rz=-126.291, fatherId=FrmDraw[0]}
  [320] = {x=-21.277, y=-8.157, z=108.914, rx=179.879, ry=0.238, rz=-125.877, fatherId=FrmDraw[0]}
  [321] = {x=-21.349, y=-8.469, z=108.908, rx=179.874, ry=0.245, rz=-125.494, fatherId=FrmDraw[0]}
  [322] = {x=-21.427, y=-8.83, z=108.901, rx=179.869, ry=0.252, rz=-125.075, fatherId=FrmDraw[0]}
  [323] = {x=-21.502, y=-9.149, z=108.894, rx=179.864, ry=0.259, rz=-124.688, fatherId=FrmDraw[0]}
  [324] = {x=-21.574, y=-9.443, z=108.888, rx=179.86, ry=0.264, rz=-124.32, fatherId=FrmDraw[0]}
  [325] = {x=-21.658, y=-9.768, z=108.882, rx=179.856, ry=0.27, rz=-123.897, fatherId=FrmDraw[0]}
  [326] = {x=-21.674, y=-9.754, z=109.374, rx=179.852, ry=0.278, rz=-123.896, fatherId=FrmDraw[0]}
  [327] = {x=-21.689, y=-9.739, z=109.866, rx=179.847, ry=0.286, rz=-123.894, fatherId=FrmDraw[0]}
  [328] = {x=-21.702, y=-9.727, z=110.259, rx=179.844, ry=0.293, rz=-123.892, fatherId=FrmDraw[0]}
  [329] = {x=-21.714, y=-9.715, z=110.653, rx=179.841, ry=0.299, rz=-123.891, fatherId=FrmDraw[0]}
  [330] = {x=-21.722, y=-9.708, z=110.888, rx=179.838, ry=0.303, rz=-123.89, fatherId=FrmDraw[0]}
  [331] = {x=-21.733, y=-9.698, z=111.243, rx=179.835, ry=0.309, rz=-123.889, fatherId=FrmDraw[0]}
  [332] = {x=-21.749, y=-9.683, z=111.722, rx=179.831, ry=0.317, rz=-123.887, fatherId=FrmDraw[0]}
  [333] = {x=-21.763, y=-9.669, z=112.17, rx=179.827, ry=0.324, rz=-123.886, fatherId=FrmDraw[0]}
  [334] = {x=-21.776, y=-9.658, z=112.552, rx=179.824, ry=0.33, rz=-123.884, fatherId=FrmDraw[0]}
  [335] = {x=-21.788, y=-9.646, z=112.935, rx=179.821, ry=0.336, rz=-123.883, fatherId=FrmDraw[0]}
  [336] = {x=-21.7, y=-9.294, z=112.942, rx=179.826, ry=0.33, rz=-124.332, fatherId=FrmDraw[0]}
  [337] = {x=-21.618, y=-8.955, z=112.948, rx=179.83, ry=0.324, rz=-124.748, fatherId=FrmDraw[0]}
  [338] = {x=-21.542, y=-8.622, z=112.955, rx=179.836, ry=0.317, rz=-125.142, fatherId=FrmDraw[0]}
  [339] = {x=-21.478, y=-8.334, z=112.96, rx=179.84, ry=0.31, rz=-125.47, fatherId=FrmDraw[0]}
  [340] = {x=-21.404, y=-8.005, z=112.967, rx=179.846, ry=0.301, rz=-125.849, fatherId=FrmDraw[0]}
  [341] = {x=-21.335, y=-7.746, z=112.974, rx=179.852, ry=0.291, rz=-126.192, fatherId=FrmDraw[0]}
  [342] = {x=-21.238, y=-7.426, z=112.982, rx=179.862, ry=0.275, rz=-126.676, fatherId=FrmDraw[0]}
  [343] = {x=-21.133, y=-7.122, z=112.992, rx=179.872, ry=0.258, rz=-127.21, fatherId=FrmDraw[0]}
  [344] = {x=-21.029, y=-6.846, z=113.001, rx=179.882, ry=0.24, rz=-127.76, fatherId=FrmDraw[0]}
  [345] = {x=-20.917, y=-6.586, z=113.01, rx=179.893, ry=0.221, rz=-128.373, fatherId=FrmDraw[0]}
  [346] = {x=-20.776, y=-6.336, z=113.022, rx=179.907, ry=0.197, rz=-129.17, fatherId=FrmDraw[0]}
  [347] = {x=-20.632, y=-6.139, z=113.033, rx=179.92, ry=0.172, rz=-130.028, fatherId=FrmDraw[0]}
  [348] = {x=-20.488, y=-5.982, z=113.043, rx=179.932, ry=0.148, rz=-130.928, fatherId=FrmDraw[0]}
  [349] = {x=-20.307, y=-5.83, z=113.055, rx=179.947, ry=0.12, rz=-132.114, fatherId=FrmDraw[0]}
  [350] = {x=-20.167, y=-5.727, z=113.065, rx=179.957, ry=0.1, rz=-133.098, fatherId=FrmDraw[0]}
  [351] = {x=-20.018, y=-5.611, z=113.074, rx=179.966, ry=0.081, rz=-134.223, fatherId=FrmDraw[0]}
  [352] = {x=-19.869, y=-5.488, z=113.083, rx=179.973, ry=0.066, rz=-135.426, fatherId=FrmDraw[0]}
  [353] = {x=-19.741, y=-5.378, z=113.09, rx=179.978, ry=0.055, rz=-136.537, fatherId=FrmDraw[0]}
  [354] = {x=-19.634, y=-5.285, z=113.096, rx=179.982, ry=0.047, rz=-137.505, fatherId=FrmDraw[0]}
  [355] = {x=-19.504, y=-5.171, z=113.103, rx=179.986, ry=0.038, rz=-138.734, fatherId=FrmDraw[0]}
  [356] = {x=-19.398, y=-5.076, z=113.108, rx=179.988, ry=0.032, rz=-139.779, fatherId=FrmDraw[0]}
  [357] = {x=-19.265, y=-4.956, z=113.115, rx=179.991, ry=0.025, rz=-141.136, fatherId=FrmDraw[0]}
  [358] = {x=-19.138, y=-4.839, z=113.121, rx=179.993, ry=0.019, rz=-142.492, fatherId=FrmDraw[0]}
  [359] = {x=-19.035, y=-4.746, z=113.126, rx=179.995, ry=0.015, rz=-143.613, fatherId=FrmDraw[0]}
  [360] = {x=-18.942, y=-4.661, z=113.13, rx=179.996, ry=0.011, rz=-144.66, fatherId=FrmDraw[0]}
  [361] = {x=-18.814, y=-4.54, z=113.136, rx=179.998, ry=0.007, rz=-146.145, fatherId=FrmDraw[0]}
  [362] = {x=-18.698, y=-4.422, z=113.142, rx=179.999, ry=0.004, rz=-147.559, fatherId=FrmDraw[0]}
  [363] = {x=-18.592, y=-4.305, z=113.146, rx=179.999, ry=0.003, rz=-148.911, fatherId=FrmDraw[0]}
  [364] = {x=-18.496, y=-4.189, z=113.15, rx=179.999, ry=0.003, rz=-150.21, fatherId=FrmDraw[0]}
  [365] = {x=-18.409, y=-4.075, z=113.154, rx=179.999, ry=0.005, rz=-151.464, fatherId=FrmDraw[0]}
  [366] = {x=-18.329, y=-3.963, z=113.157, rx=179.998, ry=0.007, rz=-152.677, fatherId=FrmDraw[0]}
  [367] = {x=-18.256, y=-3.853, z=113.16, rx=179.997, ry=0.011, rz=-153.855, fatherId=FrmDraw[0]}
  [368] = {x=-18.19, y=-3.744, z=113.162, rx=179.996, ry=0.016, rz=-155.001, fatherId=FrmDraw[0]}
  [369] = {x=-18.13, y=-3.637, z=113.164, rx=179.995, ry=0.022, rz=-156.118, fatherId=FrmDraw[0]}
  [370] = {x=-18.076, y=-3.532, z=113.165, rx=179.994, ry=0.029, rz=-157.21, fatherId=FrmDraw[0]}
  [371] = {x=-18.027, y=-3.428, z=113.166, rx=179.993, ry=0.038, rz=-158.278, fatherId=FrmDraw[0]}
  [372] = {x=-17.962, y=-3.278, z=113.167, rx=179.991, ry=0.051, rz=-159.834, fatherId=FrmDraw[0]}
  [373] = {x=-17.904, y=-3.133, z=113.167, rx=179.989, ry=0.066, rz=-161.391, fatherId=FrmDraw[0]}
  [374] = {x=-17.854, y=-2.996, z=113.167, rx=179.988, ry=0.082, rz=-162.912, fatherId=FrmDraw[0]}
  [375] = {x=-17.81, y=-2.866, z=113.167, rx=179.986, ry=0.099, rz=-164.415, fatherId=FrmDraw[0]}
  [376] = {x=-17.772, y=-2.744, z=113.166, rx=179.986, ry=0.117, rz=-165.902, fatherId=FrmDraw[0]}
  [377] = {x=-17.739, y=-2.628, z=113.165, rx=179.985, ry=0.136, rz=-167.377, fatherId=FrmDraw[0]}
  [378] = {x=-17.71, y=-2.519, z=113.163, rx=179.985, ry=0.155, rz=-168.841, fatherId=FrmDraw[0]}
  [379] = {x=-17.687, y=-2.416, z=113.161, rx=179.985, ry=0.175, rz=-170.297, fatherId=FrmDraw[0]}
  [380] = {x=-17.667, y=-2.319, z=113.159, rx=179.986, ry=0.196, rz=-171.746, fatherId=FrmDraw[0]}
  [381] = {x=-17.651, y=-2.228, z=113.156, rx=179.987, ry=0.217, rz=-173.189, fatherId=FrmDraw[0]}
  [382] = {x=-17.641, y=-2.14, z=113.153, rx=179.989, ry=0.24, rz=-174.615, fatherId=FrmDraw[0]}
  [383] = {x=-17.636, y=-2.052, z=113.15, rx=179.991, ry=0.264, rz=-176.011, fatherId=FrmDraw[0]}
  [384] = {x=-17.637, y=-1.964, z=113.146, rx=179.993, ry=0.289, rz=-177.381, fatherId=FrmDraw[0]}
  [385] = {x=-17.644, y=-1.877, z=113.142, rx=179.997, ry=0.315, rz=-178.727, fatherId=FrmDraw[0]}
  [386] = {x=-17.658, y=-1.762, z=113.136, rx=-179.999, ry=0.351, rz=179.511, fatherId=FrmDraw[0]}
  [387] = {x=-17.679, y=-1.649, z=113.129, rx=-179.992, ry=0.387, rz=177.778, fatherId=FrmDraw[0]}
  [388] = {x=-17.703, y=-1.541, z=113.123, rx=-179.985, ry=0.423, rz=176.057, fatherId=FrmDraw[0]}
  [389] = {x=-17.728, y=-1.439, z=113.116, rx=-179.977, ry=0.458, rz=174.342, fatherId=FrmDraw[0]}
  [390] = {x=-17.753, y=-1.343, z=113.11, rx=-179.968, ry=0.491, rz=172.631, fatherId=FrmDraw[0]}
  [391] = {x=-17.776, y=-1.253, z=113.104, rx=-179.959, ry=0.521, rz=170.92, fatherId=FrmDraw[0]}
  [392] = {x=-17.798, y=-1.163, z=113.098, rx=-179.948, ry=0.549, rz=169.233, fatherId=FrmDraw[0]}
  [393] = {x=-17.824, y=-1.065, z=113.092, rx=-179.937, ry=0.576, rz=167.61, fatherId=FrmDraw[0]}
  [394] = {x=-17.854, y=-0.958, z=113.086, rx=-179.926, ry=0.604, rz=166.047, fatherId=FrmDraw[0]}
  [395] = {x=-17.888, y=-0.842, z=113.08, rx=-179.914, ry=0.631, rz=164.543, fatherId=FrmDraw[0]}
  [396] = {x=-17.926, y=-0.719, z=113.074, rx=-179.902, ry=0.658, rz=163.093, fatherId=FrmDraw[0]}
  [397] = {x=-17.97, y=-0.588, z=113.068, rx=-179.89, ry=0.686, rz=161.695, fatherId=FrmDraw[0]}
  [398] = {x=-18.018, y=-0.449, z=113.061, rx=-179.876, ry=0.714, rz=160.347, fatherId=FrmDraw[0]}
  [399] = {x=-18.072, y=-0.304, z=113.054, rx=-179.863, ry=0.742, rz=159.044, fatherId=FrmDraw[0]}
  [400] = {x=-18.131, y=-0.153, z=113.047, rx=-179.849, ry=0.771, rz=157.785, fatherId=FrmDraw[0]}
  [401] = {x=-18.195, y=0.005, z=113.039, rx=-179.834, ry=0.801, rz=156.567, fatherId=FrmDraw[0]}
  [402] = {x=-18.263, y=0.165, z=113.032, rx=-179.819, ry=0.831, rz=155.371, fatherId=FrmDraw[0]}
  [403] = {x=-18.334, y=0.321, z=113.024, rx=-179.803, ry=0.861, rz=154.168, fatherId=FrmDraw[0]}
  [404] = {x=-18.408, y=0.474, z=113.016, rx=-179.786, ry=0.89, rz=152.956, fatherId=FrmDraw[0]}
  [405] = {x=-18.485, y=0.622, z=113.009, rx=-179.769, ry=0.918, rz=151.735, fatherId=FrmDraw[0]}
  [406] = {x=-18.565, y=0.767, z=113.001, rx=-179.751, ry=0.946, rz=150.504, fatherId=FrmDraw[0]}
  [407] = {x=-18.647, y=0.908, z=112.994, rx=-179.733, ry=0.973, rz=149.26, fatherId=FrmDraw[0]}
  [408] = {x=-18.734, y=1.044, z=112.986, rx=-179.713, ry=1, rz=148.003, fatherId=FrmDraw[0]}
  [409] = {x=-18.823, y=1.175, z=112.978, rx=-179.693, ry=1.026, rz=146.732, fatherId=FrmDraw[0]}
  [410] = {x=-18.917, y=1.301, z=112.97, rx=-179.673, ry=1.052, rz=145.445, fatherId=FrmDraw[0]}
  [411] = {x=-19.014, y=1.423, z=112.962, rx=-179.651, ry=1.078, rz=144.141, fatherId=FrmDraw[0]}
  [412] = {x=-19.115, y=1.541, z=112.954, rx=-179.629, ry=1.104, rz=142.831, fatherId=FrmDraw[0]}
  [413] = {x=-19.222, y=1.664, z=112.945, rx=-179.605, ry=1.132, rz=141.553, fatherId=FrmDraw[0]}
  [414] = {x=-19.306, y=1.761, z=112.939, rx=-179.587, ry=1.153, rz=140.619, fatherId=FrmDraw[0]}
  [415] = {x=-19.42, y=1.896, z=112.93, rx=-179.563, ry=1.183, rz=139.405, fatherId=FrmDraw[0]}
  [416] = {x=-19.538, y=2.038, z=112.92, rx=-179.537, ry=1.213, rz=138.227, fatherId=FrmDraw[0]}
  [417] = {x=-19.659, y=2.188, z=112.911, rx=-179.511, ry=1.243, rz=137.085, fatherId=FrmDraw[0]}
  [418] = {x=-19.782, y=2.346, z=112.901, rx=-179.485, ry=1.274, rz=135.98, fatherId=FrmDraw[0]}
  [419] = {x=-19.906, y=2.512, z=112.892, rx=-179.459, ry=1.304, rz=134.91, fatherId=FrmDraw[0]}
  [420] = {x=-20.03, y=2.687, z=112.883, rx=-179.432, ry=1.333, rz=133.875, fatherId=FrmDraw[0]}
  [421] = {x=-20.153, y=2.871, z=112.874, rx=-179.407, ry=1.361, rz=132.874, fatherId=FrmDraw[0]}
  [422] = {x=-20.275, y=3.065, z=112.865, rx=-179.381, ry=1.387, rz=131.906, fatherId=FrmDraw[0]}
  [423] = {x=-20.394, y=3.266, z=112.858, rx=-179.357, ry=1.41, rz=130.954, fatherId=FrmDraw[0]}
  [424] = {x=-20.513, y=3.471, z=112.851, rx=-179.333, ry=1.432, rz=130.012, fatherId=FrmDraw[0]}
  [425] = {x=-20.631, y=3.682, z=112.844, rx=-179.309, ry=1.451, rz=129.082, fatherId=FrmDraw[0]}
  [426] = {x=-20.75, y=3.897, z=112.837, rx=-179.286, ry=1.469, rz=128.163, fatherId=FrmDraw[0]}
  [427] = {x=-20.863, y=4.107, z=112.832, rx=-179.264, ry=1.486, rz=127.301, fatherId=FrmDraw[0]}
  [428] = {x=-20.984, y=4.331, z=112.826, rx=-179.241, ry=1.502, rz=126.403, fatherId=FrmDraw[0]}
  [429] = {x=-21.108, y=4.56, z=112.82, rx=-179.218, ry=1.518, rz=125.516, fatherId=FrmDraw[0]}
  [430] = {x=-21.236, y=4.793, z=112.814, rx=-179.195, ry=1.534, rz=124.64, fatherId=FrmDraw[0]}
  [431] = {x=-21.367, y=5.029, z=112.808, rx=-179.171, ry=1.551, rz=123.774, fatherId=FrmDraw[0]}
  [432] = {x=-21.503, y=5.271, z=112.802, rx=-179.147, ry=1.569, rz=122.93, fatherId=FrmDraw[0]}
  [433] = {x=-21.642, y=5.523, z=112.795, rx=-179.121, ry=1.589, rz=122.126, fatherId=FrmDraw[0]}
  [434] = {x=-21.782, y=5.786, z=112.789, rx=-179.096, ry=1.61, rz=121.362, fatherId=FrmDraw[0]}
  [435] = {x=-21.922, y=6.061, z=112.783, rx=-179.07, ry=1.632, rz=120.639, fatherId=FrmDraw[0]}
  [436] = {x=-22.061, y=6.347, z=112.777, rx=-179.044, ry=1.654, rz=119.962, fatherId=FrmDraw[0]}
  [437] = {x=-22.194, y=6.64, z=112.771, rx=-179.02, ry=1.676, rz=119.341, fatherId=FrmDraw[0]}
  [438] = {x=-22.306, y=6.903, z=112.767, rx=-178.999, ry=1.694, rz=118.842, fatherId=FrmDraw[0]}
  [439] = {x=-22.396, y=7.129, z=112.763, rx=-178.983, ry=1.708, rz=118.45, fatherId=FrmDraw[0]}
  [440] = {x=-22.516, y=7.46, z=112.759, rx=-178.961, ry=1.727, rz=117.939, fatherId=FrmDraw[0]}
  [441] = {x=-22.614, y=7.756, z=112.756, rx=-178.943, ry=1.742, rz=117.533, fatherId=FrmDraw[0]}
  [442] = {x=-22.689, y=7.999, z=112.754, rx=-178.931, ry=1.753, rz=117.223, fatherId=FrmDraw[0]}
  [443] = {x=-22.778, y=8.311, z=112.753, rx=-178.916, ry=1.764, rz=116.853, fatherId=FrmDraw[0]}
  [444] = {x=-22.846, y=8.567, z=112.752, rx=-178.904, ry=1.773, rz=116.571, fatherId=FrmDraw[0]}
  [445] = {x=-22.929, y=8.894, z=112.751, rx=-178.891, ry=1.782, rz=116.235, fatherId=FrmDraw[0]}
  [446] = {x=-22.991, y=9.162, z=112.75, rx=-178.882, ry=1.789, rz=115.981, fatherId=FrmDraw[0]}
  [447] = {x=-23.067, y=9.504, z=112.75, rx=-178.87, ry=1.797, rz=115.682, fatherId=FrmDraw[0]}
  [448] = {x=-23.125, y=9.783, z=112.75, rx=-178.862, ry=1.802, rz=115.457, fatherId=FrmDraw[0]}
  [449] = {x=-23.194, y=10.139, z=112.751, rx=-178.852, ry=1.809, rz=115.195, fatherId=FrmDraw[0]}
  [450] = {x=-23.248, y=10.429, z=112.751, rx=-178.844, ry=1.815, rz=115, fatherId=FrmDraw[0]}
  [451] = {x=-23.312, y=10.798, z=112.752, rx=-178.834, ry=1.822, rz=114.775, fatherId=FrmDraw[0]}
  [452] = {x=-23.368, y=11.135, z=112.753, rx=-178.826, ry=1.828, rz=114.59, fatherId=FrmDraw[0]}
  [453] = {x=-23.424, y=11.474, z=112.754, rx=-178.818, ry=1.835, rz=114.406, fatherId=FrmDraw[0]}
  [454] = {x=-23.482, y=11.814, z=112.755, rx=-178.809, ry=1.841, rz=114.219, fatherId=FrmDraw[0]}
  [455] = {x=-23.541, y=12.153, z=112.756, rx=-178.801, ry=1.847, rz=114.031, fatherId=FrmDraw[0]}
  [456] = {x=-23.601, y=12.493, z=112.757, rx=-178.793, ry=1.853, rz=113.841, fatherId=FrmDraw[0]}
  [457] = {x=-23.662, y=12.834, z=112.759, rx=-178.785, ry=1.858, rz=113.649, fatherId=FrmDraw[0]}
  [458] = {x=-23.725, y=13.175, z=112.76, rx=-178.777, ry=1.864, rz=113.454, fatherId=FrmDraw[0]}
  [459] = {x=-23.789, y=13.516, z=112.761, rx=-178.769, ry=1.869, rz=113.257, fatherId=FrmDraw[0]}
  [460] = {x=-23.848, y=13.82, z=112.763, rx=-178.762, ry=1.874, rz=113.081, fatherId=FrmDraw[0]}
  [461] = {x=-23.922, y=14.2, z=112.764, rx=-178.753, ry=1.879, rz=112.857, fatherId=FrmDraw[0]}
  [462] = {x=-23.983, y=14.504, z=112.766, rx=-178.746, ry=1.883, rz=112.677, fatherId=FrmDraw[0]}
  [463] = {x=-24.061, y=14.885, z=112.768, rx=-178.737, ry=1.888, rz=112.448, fatherId=FrmDraw[0]}
  [464] = {x=-24.125, y=15.191, z=112.769, rx=-178.73, ry=1.892, rz=112.263, fatherId=FrmDraw[0]}
  [465] = {x=-24.207, y=15.573, z=112.771, rx=-178.722, ry=1.896, rz=112.03, fatherId=FrmDraw[0]}
  [466] = {x=-24.273, y=15.879, z=112.773, rx=-178.715, ry=1.899, rz=111.841, fatherId=FrmDraw[0]}
  [467] = {x=-24.359, y=16.262, z=112.775, rx=-178.707, ry=1.903, rz=111.602, fatherId=FrmDraw[0]}
  [468] = {x=-24.428, y=16.569, z=112.777, rx=-178.7, ry=1.906, rz=111.408, fatherId=FrmDraw[0]}
  [469] = {x=-24.518, y=16.953, z=112.779, rx=-178.692, ry=1.91, rz=111.164, fatherId=FrmDraw[0]}
  [470] = {x=-24.591, y=17.261, z=112.781, rx=-178.685, ry=1.912, rz=110.966, fatherId=FrmDraw[0]}
  [471] = {x=-24.684, y=17.646, z=112.783, rx=-178.677, ry=1.915, rz=110.716, fatherId=FrmDraw[0]}
  [472] = {x=-24.761, y=17.954, z=112.785, rx=-178.67, ry=1.918, rz=110.513, fatherId=FrmDraw[0]}
  [473] = {x=-24.858, y=18.341, z=112.787, rx=-178.662, ry=1.92, rz=110.257, fatherId=FrmDraw[0]}
  [474] = {x=-24.938, y=18.651, z=112.789, rx=-178.655, ry=1.922, rz=110.053, fatherId=FrmDraw[0]}
  [475] = {x=-25.036, y=19.042, z=112.792, rx=-178.647, ry=1.925, rz=109.803, fatherId=FrmDraw[0]}
  [476] = {x=-25.125, y=19.396, z=112.794, rx=-178.64, ry=1.927, rz=109.583, fatherId=FrmDraw[0]}
  [477] = {x=-25.213, y=19.753, z=112.797, rx=-178.633, ry=1.929, rz=109.368, fatherId=FrmDraw[0]}
  [478] = {x=-25.301, y=20.113, z=112.799, rx=-178.626, ry=1.932, rz=109.158, fatherId=FrmDraw[0]}
  [479] = {x=-25.388, y=20.475, z=112.802, rx=-178.619, ry=1.934, rz=108.952, fatherId=FrmDraw[0]}
  [480] = {x=-25.475, y=20.84, z=112.805, rx=-178.612, ry=1.937, rz=108.752, fatherId=FrmDraw[0]}
  [481] = {x=-25.561, y=21.208, z=112.808, rx=-178.605, ry=1.939, rz=108.556, fatherId=FrmDraw[0]}
  [482] = {x=-25.646, y=21.578, z=112.811, rx=-178.599, ry=1.942, rz=108.366, fatherId=FrmDraw[0]}
  [483] = {x=-25.731, y=21.951, z=112.814, rx=-178.592, ry=1.945, rz=108.181, fatherId=FrmDraw[0]}
  [484] = {x=-25.806, y=22.284, z=112.816, rx=-178.586, ry=1.947, rz=108.017, fatherId=FrmDraw[0]}
  [485] = {x=-25.904, y=22.699, z=112.82, rx=-178.578, ry=1.95, rz=107.807, fatherId=FrmDraw[0]}
  [486] = {x=-25.985, y=23.031, z=112.823, rx=-178.573, ry=1.951, rz=107.633, fatherId=FrmDraw[0]}
  [487] = {x=-26.09, y=23.446, z=112.826, rx=-178.566, ry=1.953, rz=107.408, fatherId=FrmDraw[0]}
  [488] = {x=-26.176, y=23.779, z=112.829, rx=-178.561, ry=1.953, rz=107.222, fatherId=FrmDraw[0]}
  [489] = {x=-26.285, y=24.194, z=112.833, rx=-178.555, ry=1.952, rz=106.983, fatherId=FrmDraw[0]}
  [490] = {x=-26.394, y=24.598, z=112.836, rx=-178.551, ry=1.949, rz=106.744, fatherId=FrmDraw[0]}
  [491] = {x=-26.489, y=24.946, z=112.839, rx=-178.548, ry=1.945, rz=106.532, fatherId=FrmDraw[0]}
  [492] = {x=-26.6, y=25.352, z=112.842, rx=-178.546, ry=1.939, rz=106.279, fatherId=FrmDraw[0]}
  [493] = {x=-26.732, y=25.679, z=112.844, rx=-178.545, ry=1.93, rz=105.976, fatherId=FrmDraw[0]}
  [494] = {x=-26.728, y=25.68, z=113.344, rx=-178.545, ry=1.931, rz=105.987, fatherId=FrmDraw[0]}
  [495] = {x=-26.724, y=25.682, z=113.844, rx=-178.544, ry=1.931, rz=105.998, fatherId=FrmDraw[0]}
  [496] = {x=-26.721, y=25.683, z=114.244, rx=-178.544, ry=1.932, rz=106.007, fatherId=FrmDraw[0]}
  [497] = {x=-26.718, y=25.684, z=114.644, rx=-178.544, ry=1.933, rz=106.016, fatherId=FrmDraw[0]}
  [498] = {x=-26.716, y=25.685, z=114.883, rx=-178.544, ry=1.933, rz=106.021, fatherId=FrmDraw[0]}
  [499] = {x=-26.713, y=25.686, z=115.244, rx=-178.544, ry=1.934, rz=106.029, fatherId=FrmDraw[0]}
  [500] = {x=-26.71, y=25.687, z=115.719, rx=-178.543, ry=1.935, rz=106.04, fatherId=FrmDraw[0]}
  [501] = {x=-26.706, y=25.689, z=116.169, rx=-178.543, ry=1.935, rz=106.05, fatherId=FrmDraw[0]}
  [502] = {x=-26.703, y=25.69, z=116.538, rx=-178.543, ry=1.936, rz=106.058, fatherId=FrmDraw[0]}
  [503] = {x=-26.7, y=25.691, z=116.907, rx=-178.542, ry=1.936, rz=106.066, fatherId=FrmDraw[0]}
  [504] = {x=-26.604, y=25.339, z=116.904, rx=-178.541, ry=1.947, rz=106.303, fatherId=FrmDraw[0]}
  [505] = {x=-26.507, y=24.922, z=116.9, rx=-178.541, ry=1.955, rz=106.534, fatherId=FrmDraw[0]}
  [506] = {x=-26.422, y=24.567, z=116.897, rx=-178.543, ry=1.959, rz=106.73, fatherId=FrmDraw[0]}
  [507] = {x=-26.321, y=24.159, z=116.893, rx=-178.547, ry=1.962, rz=106.952, fatherId=FrmDraw[0]}
  [508] = {x=-26.215, y=23.739, z=116.89, rx=-178.553, ry=1.962, rz=107.177, fatherId=FrmDraw[0]}
  [509] = {x=-26.131, y=23.406, z=116.887, rx=-178.558, ry=1.961, rz=107.354, fatherId=FrmDraw[0]}
  [510] = {x=-26.026, y=22.991, z=116.883, rx=-178.566, ry=1.958, rz=107.571, fatherId=FrmDraw[0]}
  [511] = {x=-25.944, y=22.659, z=116.88, rx=-178.573, ry=1.955, rz=107.742, fatherId=FrmDraw[0]}
  [512] = {x=-25.844, y=22.245, z=116.877, rx=-178.581, ry=1.951, rz=107.95, fatherId=FrmDraw[0]}
  [513] = {x=-25.766, y=21.914, z=116.874, rx=-178.587, ry=1.948, rz=108.114, fatherId=FrmDraw[0]}
  [514] = {x=-25.67, y=21.501, z=116.871, rx=-178.595, ry=1.945, rz=108.322, fatherId=FrmDraw[0]}
  [515] = {x=-25.594, y=21.173, z=116.868, rx=-178.601, ry=1.943, rz=108.493, fatherId=FrmDraw[0]}
  [516] = {x=-25.498, y=20.764, z=116.865, rx=-178.609, ry=1.94, rz=108.712, fatherId=FrmDraw[0]}
  [517] = {x=-25.421, y=20.44, z=116.863, rx=-178.614, ry=1.938, rz=108.891, fatherId=FrmDraw[0]}
  [518] = {x=-25.325, y=20.036, z=116.859, rx=-178.622, ry=1.937, rz=109.119, fatherId=FrmDraw[0]}
  [519] = {x=-25.249, y=19.716, z=116.857, rx=-178.627, ry=1.935, rz=109.307, fatherId=FrmDraw[0]}
  [520] = {x=-25.153, y=19.318, z=116.854, rx=-178.635, ry=1.934, rz=109.545, fatherId=FrmDraw[0]}
  [521] = {x=-25.075, y=19.002, z=116.852, rx=-178.64, ry=1.932, rz=109.74, fatherId=FrmDraw[0]}
  [522] = {x=-24.979, y=18.61, z=116.849, rx=-178.648, ry=1.931, rz=109.989, fatherId=FrmDraw[0]}
  [523] = {x=-24.901, y=18.298, z=116.847, rx=-178.654, ry=1.929, rz=110.192, fatherId=FrmDraw[0]}
  [524] = {x=-24.805, y=17.911, z=116.845, rx=-178.662, ry=1.927, rz=110.445, fatherId=FrmDraw[0]}
  [525] = {x=-24.729, y=17.601, z=116.843, rx=-178.668, ry=1.925, rz=110.646, fatherId=FrmDraw[0]}
  [526] = {x=-24.636, y=17.216, z=116.84, rx=-178.676, ry=1.923, rz=110.894, fatherId=FrmDraw[0]}
  [527] = {x=-24.563, y=16.907, z=116.838, rx=-178.683, ry=1.92, rz=111.09, fatherId=FrmDraw[0]}
  [528] = {x=-24.474, y=16.523, z=116.836, rx=-178.691, ry=1.916, rz=111.332, fatherId=FrmDraw[0]}
  [529] = {x=-24.404, y=16.216, z=116.834, rx=-178.698, ry=1.913, rz=111.524, fatherId=FrmDraw[0]}
  [530] = {x=-24.319, y=15.833, z=116.832, rx=-178.706, ry=1.909, rz=111.76, fatherId=FrmDraw[0]}
  [531] = {x=-24.251, y=15.527, z=116.831, rx=-178.713, ry=1.905, rz=111.948, fatherId=FrmDraw[0]}
  [532] = {x=-24.169, y=15.145, z=116.829, rx=-178.722, ry=1.901, rz=112.179, fatherId=FrmDraw[0]}
  [533] = {x=-24.105, y=14.84, z=116.827, rx=-178.729, ry=1.896, rz=112.363, fatherId=FrmDraw[0]}
  [534] = {x=-24.026, y=14.459, z=116.825, rx=-178.738, ry=1.891, rz=112.589, fatherId=FrmDraw[0]}
  [535] = {x=-23.964, y=14.155, z=116.824, rx=-178.746, ry=1.887, rz=112.768, fatherId=FrmDraw[0]}
  [536] = {x=-23.888, y=13.775, z=116.822, rx=-178.755, ry=1.881, rz=112.99, fatherId=FrmDraw[0]}
  [537] = {x=-23.829, y=13.472, z=116.821, rx=-178.762, ry=1.876, rz=113.165, fatherId=FrmDraw[0]}
  [538] = {x=-23.756, y=13.093, z=116.819, rx=-178.771, ry=1.87, rz=113.382, fatherId=FrmDraw[0]}
  [539] = {x=-23.699, y=12.79, z=116.818, rx=-178.779, ry=1.864, rz=113.553, fatherId=FrmDraw[0]}
  [540] = {x=-23.63, y=12.413, z=116.817, rx=-178.788, ry=1.858, rz=113.765, fatherId=FrmDraw[0]}
  [541] = {x=-23.576, y=12.111, z=116.816, rx=-178.796, ry=1.852, rz=113.933, fatherId=FrmDraw[0]}
  [542] = {x=-23.509, y=11.733, z=116.815, rx=-178.805, ry=1.845, rz=114.141, fatherId=FrmDraw[0]}
  [543] = {x=-23.458, y=11.432, z=116.814, rx=-178.812, ry=1.839, rz=114.305, fatherId=FrmDraw[0]}
  [544] = {x=-23.394, y=11.056, z=116.813, rx=-178.822, ry=1.832, rz=114.508, fatherId=FrmDraw[0]}
  [545] = {x=-23.344, y=10.756, z=116.812, rx=-178.829, ry=1.826, rz=114.673, fatherId=FrmDraw[0]}
  [546] = {x=-23.28, y=10.387, z=116.811, rx=-178.839, ry=1.819, rz=114.897, fatherId=FrmDraw[0]}
  [547] = {x=-23.226, y=10.096, z=116.81, rx=-178.846, ry=1.814, rz=115.089, fatherId=FrmDraw[0]}
  [548] = {x=-23.157, y=9.739, z=116.81, rx=-178.857, ry=1.807, rz=115.346, fatherId=FrmDraw[0]}
  [549] = {x=-23.1, y=9.458, z=116.81, rx=-178.865, ry=1.801, rz=115.564, fatherId=FrmDraw[0]}
  [550] = {x=-23.025, y=9.114, z=116.81, rx=-178.876, ry=1.793, rz=115.854, fatherId=FrmDraw[0]}
  [551] = {x=-22.963, y=8.844, z=116.81, rx=-178.886, ry=1.786, rz=116.098, fatherId=FrmDraw[0]}
  [552] = {x=-22.882, y=8.513, z=116.811, rx=-178.899, ry=1.776, rz=116.419, fatherId=FrmDraw[0]}
  [553] = {x=-22.814, y=8.255, z=116.812, rx=-178.91, ry=1.767, rz=116.689, fatherId=FrmDraw[0]}
  [554] = {x=-22.725, y=7.939, z=116.814, rx=-178.925, ry=1.755, rz=117.041, fatherId=FrmDraw[0]}
  [555] = {x=-22.651, y=7.692, z=116.816, rx=-178.938, ry=1.744, rz=117.335, fatherId=FrmDraw[0]}
  [556] = {x=-22.553, y=7.392, z=116.819, rx=-178.956, ry=1.728, rz=117.72, fatherId=FrmDraw[0]}
  [557] = {x=-22.432, y=7.057, z=116.823, rx=-178.978, ry=1.707, rz=118.214, fatherId=FrmDraw[0]}
  [558] = {x=-22.341, y=6.829, z=116.826, rx=-178.995, ry=1.692, rz=118.596, fatherId=FrmDraw[0]}
  [559] = {x=-22.228, y=6.565, z=116.831, rx=-179.016, ry=1.674, rz=119.085, fatherId=FrmDraw[0]}
  [560] = {x=-22.093, y=6.271, z=116.837, rx=-179.041, ry=1.651, rz=119.699, fatherId=FrmDraw[0]}
  [561] = {x=-21.995, y=6.07, z=116.841, rx=-179.059, ry=1.636, rz=120.165, fatherId=FrmDraw[0]}
  [562] = {x=-21.877, y=5.837, z=116.846, rx=-179.081, ry=1.617, rz=120.755, fatherId=FrmDraw[0]}
  [563] = {x=-21.738, y=5.577, z=116.852, rx=-179.106, ry=1.596, rz=121.483, fatherId=FrmDraw[0]}
  [564] = {x=-21.597, y=5.323, z=116.859, rx=-179.131, ry=1.576, rz=122.272, fatherId=FrmDraw[0]}
  [565] = {x=-21.458, y=5.079, z=116.865, rx=-179.156, ry=1.557, rz=123.108, fatherId=FrmDraw[0]}
  [566] = {x=-21.323, y=4.843, z=116.871, rx=-179.18, ry=1.541, rz=123.977, fatherId=FrmDraw[0]}
  [567] = {x=-21.193, y=4.61, z=116.877, rx=-179.204, ry=1.525, rz=124.853, fatherId=FrmDraw[0]}
  [568] = {x=-21.066, y=4.38, z=116.883, rx=-179.227, ry=1.509, rz=125.736, fatherId=FrmDraw[0]}
  [569] = {x=-20.943, y=4.153, z=116.889, rx=-179.25, ry=1.492, rz=126.626, fatherId=FrmDraw[0]}
  [570] = {x=-20.822, y=3.929, z=116.895, rx=-179.273, ry=1.476, rz=127.524, fatherId=FrmDraw[0]}
  [571] = {x=-20.702, y=3.71, z=116.901, rx=-179.296, ry=1.458, rz=128.429, fatherId=FrmDraw[0]}
  [572] = {x=-20.583, y=3.494, z=116.908, rx=-179.319, ry=1.438, rz=129.342, fatherId=FrmDraw[0]}
  [573] = {x=-20.469, y=3.294, z=116.914, rx=-179.342, ry=1.418, rz=130.216, fatherId=FrmDraw[0]}
  [574] = {x=-20.348, y=3.088, z=116.922, rx=-179.366, ry=1.395, rz=131.144, fatherId=FrmDraw[0]}
  [575] = {x=-20.226, y=2.886, z=116.93, rx=-179.392, ry=1.369, rz=132.081, fatherId=FrmDraw[0]}
  [576] = {x=-20.102, y=2.694, z=116.939, rx=-179.418, ry=1.341, rz=133.05, fatherId=FrmDraw[0]}
  [577] = {x=-19.976, y=2.513, z=116.948, rx=-179.444, ry=1.312, rz=134.057, fatherId=FrmDraw[0]}
  [578] = {x=-19.851, y=2.342, z=116.957, rx=-179.47, ry=1.283, rz=135.104, fatherId=FrmDraw[0]}
  [579] = {x=-19.727, y=2.18, z=116.967, rx=-179.496, ry=1.252, rz=136.189, fatherId=FrmDraw[0]}
  [580] = {x=-19.605, y=2.027, z=116.976, rx=-179.522, ry=1.222, rz=137.314, fatherId=FrmDraw[0]}
  [581] = {x=-19.485, y=1.882, z=116.986, rx=-179.548, ry=1.192, rz=138.478, fatherId=FrmDraw[0]}
  [582] = {x=-19.397, y=1.779, z=116.993, rx=-179.567, ry=1.17, rz=139.378, fatherId=FrmDraw[0]}
  [583] = {x=-19.311, y=1.68, z=116.999, rx=-179.585, ry=1.149, rz=140.3, fatherId=FrmDraw[0]}
  [584] = {x=-19.201, y=1.555, z=117.008, rx=-179.609, ry=1.121, rz=141.564, fatherId=FrmDraw[0]}
  [585] = {x=-19.096, y=1.436, z=117.016, rx=-179.632, ry=1.095, rz=142.867, fatherId=FrmDraw[0]}
  [586] = {x=-18.996, y=1.319, z=117.024, rx=-179.654, ry=1.07, rz=144.186, fatherId=FrmDraw[0]}
  [587] = {x=-18.9, y=1.197, z=117.032, rx=-179.676, ry=1.044, rz=145.487, fatherId=FrmDraw[0]}
  [588] = {x=-18.806, y=1.07, z=117.04, rx=-179.696, ry=1.018, rz=146.77, fatherId=FrmDraw[0]}
  [589] = {x=-18.717, y=0.938, z=117.048, rx=-179.716, ry=0.992, rz=148.037, fatherId=FrmDraw[0]}
  [590] = {x=-18.631, y=0.802, z=117.056, rx=-179.735, ry=0.965, rz=149.29, fatherId=FrmDraw[0]}
  [591] = {x=-18.548, y=0.66, z=117.063, rx=-179.753, ry=0.937, rz=150.529, fatherId=FrmDraw[0]}
  [592] = {x=-18.468, y=0.515, z=117.071, rx=-179.771, ry=0.91, rz=151.756, fatherId=FrmDraw[0]}
  [593] = {x=-18.391, y=0.365, z=117.078, rx=-179.788, ry=0.881, rz=152.972, fatherId=FrmDraw[0]}
  [594] = {x=-18.318, y=0.211, z=117.086, rx=-179.805, ry=0.853, rz=154.178, fatherId=FrmDraw[0]}
  [595] = {x=-18.247, y=0.054, z=117.094, rx=-179.82, ry=0.824, rz=155.376, fatherId=FrmDraw[0]}
  [596] = {x=-18.181, y=-0.105, z=117.101, rx=-179.835, ry=0.794, rz=156.577, fatherId=FrmDraw[0]}
  [597] = {x=-18.12, y=-0.259, z=117.108, rx=-179.85, ry=0.766, rz=157.814, fatherId=FrmDraw[0]}
  [598] = {x=-18.065, y=-0.407, z=117.115, rx=-179.864, ry=0.739, rz=159.092, fatherId=FrmDraw[0]}
  [599] = {x=-18.015, y=-0.548, z=117.121, rx=-179.877, ry=0.712, rz=160.413, fatherId=FrmDraw[0]}
  [600] = {x=-17.97, y=-0.683, z=117.128, rx=-179.89, ry=0.685, rz=161.779, fatherId=FrmDraw[0]}
  [601] = {x=-17.929, y=-0.811, z=117.134, rx=-179.903, ry=0.659, rz=163.193, fatherId=FrmDraw[0]}
  [602] = {x=-17.893, y=-0.932, z=117.14, rx=-179.915, ry=0.633, rz=164.657, fatherId=FrmDraw[0]}
  [603] = {x=-17.86, y=-1.044, z=117.146, rx=-179.927, ry=0.606, rz=166.175, fatherId=FrmDraw[0]}
  [604] = {x=-17.831, y=-1.149, z=117.152, rx=-179.938, ry=0.579, rz=167.75, fatherId=FrmDraw[0]}
  [605] = {x=-17.804, y=-1.245, z=117.158, rx=-179.949, ry=0.55, rz=169.383, fatherId=FrmDraw[0]}
  [606] = {x=-17.778, y=-1.336, z=117.164, rx=-179.959, ry=0.52, rz=171.064, fatherId=FrmDraw[0]}
  [607] = {x=-17.748, y=-1.431, z=117.17, rx=-179.969, ry=0.487, rz=172.752, fatherId=FrmDraw[0]}
  [608] = {x=-17.718, y=-1.53, z=117.177, rx=-179.978, ry=0.452, rz=174.448, fatherId=FrmDraw[0]}
  [609] = {x=-17.689, y=-1.634, z=117.184, rx=-179.986, ry=0.415, rz=176.154, fatherId=FrmDraw[0]}
  [610] = {x=-17.663, y=-1.742, z=117.191, rx=-179.993, ry=0.378, rz=177.876, fatherId=FrmDraw[0]}
  [611] = {x=-17.643, y=-1.853, z=117.198, rx=-179.999, ry=0.341, rz=179.622, fatherId=FrmDraw[0]}
  [612] = {x=-17.631, y=-1.964, z=117.204, rx=179.996, ry=0.306, rz=-178.596, fatherId=FrmDraw[0]}
  [613] = {x=-17.627, y=-2.048, z=117.208, rx=179.993, ry=0.281, rz=-177.232, fatherId=FrmDraw[0]}
  [614] = {x=-17.63, y=-2.132, z=117.211, rx=179.991, ry=0.257, rz=-175.841, fatherId=FrmDraw[0]}
  [615] = {x=-17.639, y=-2.215, z=117.214, rx=179.989, ry=0.235, rz=-174.421, fatherId=FrmDraw[0]}
  [616] = {x=-17.653, y=-2.3, z=117.217, rx=179.987, ry=0.214, rz=-172.976, fatherId=FrmDraw[0]}
  [617] = {x=-17.671, y=-2.39, z=117.219, rx=179.986, ry=0.194, rz=-171.526, fatherId=FrmDraw[0]}
  [618] = {x=-17.693, y=-2.486, z=117.221, rx=179.985, ry=0.174, rz=-170.07, fatherId=FrmDraw[0]}
  [619] = {x=-17.72, y=-2.588, z=117.223, rx=179.985, ry=0.154, rz=-168.606, fatherId=FrmDraw[0]}
  [620] = {x=-17.75, y=-2.696, z=117.225, rx=179.985, ry=0.136, rz=-167.134, fatherId=FrmDraw[0]}
  [621] = {x=-17.785, y=-2.811, z=117.226, rx=179.985, ry=0.118, rz=-165.65, fatherId=FrmDraw[0]}
  [622] = {x=-17.826, y=-2.933, z=117.226, rx=179.986, ry=0.101, rz=-164.153, fatherId=FrmDraw[0]}
  [623] = {x=-17.872, y=-3.061, z=117.227, rx=179.987, ry=0.084, rz=-162.639, fatherId=FrmDraw[0]}
  [624] = {x=-17.925, y=-3.196, z=117.226, rx=179.989, ry=0.069, rz=-161.112, fatherId=FrmDraw[0]}
  [625] = {x=-17.985, y=-3.339, z=117.226, rx=179.99, ry=0.054, rz=-159.547, fatherId=FrmDraw[0]}
  [626] = {x=-18.052, y=-3.484, z=117.225, rx=179.992, ry=0.042, rz=-157.989, fatherId=FrmDraw[0]}
  [627] = {x=-18.103, y=-3.584, z=117.223, rx=179.993, ry=0.034, rz=-156.914, fatherId=FrmDraw[0]}
  [628] = {x=-18.16, y=-3.686, z=117.222, rx=179.994, ry=0.028, rz=-155.815, fatherId=FrmDraw[0]}
  [629] = {x=-18.222, y=-3.789, z=117.22, rx=179.995, ry=0.022, rz=-154.691, fatherId=FrmDraw[0]}
  [630] = {x=-18.29, y=-3.893, z=117.218, rx=179.996, ry=0.017, rz=-153.539, fatherId=FrmDraw[0]}
  [631] = {x=-18.365, y=-3.999, z=117.215, rx=179.997, ry=0.014, rz=-152.355, fatherId=FrmDraw[0]}
  [632] = {x=-18.446, y=-4.107, z=117.212, rx=179.997, ry=0.011, rz=-151.136, fatherId=FrmDraw[0]}
  [633] = {x=-18.535, y=-4.216, z=117.208, rx=179.997, ry=0.01, rz=-149.877, fatherId=FrmDraw[0]}
  [634] = {x=-18.633, y=-4.327, z=117.204, rx=179.997, ry=0.01, rz=-148.573, fatherId=FrmDraw[0]}
  [635] = {x=-18.74, y=-4.439, z=117.199, rx=179.996, ry=0.012, rz=-147.217, fatherId=FrmDraw[0]}
  [636] = {x=-18.858, y=-4.553, z=117.194, rx=179.995, ry=0.015, rz=-145.799, fatherId=FrmDraw[0]}
  [637] = {x=-18.988, y=-4.669, z=117.188, rx=179.994, ry=0.02, rz=-144.312, fatherId=FrmDraw[0]}
  [638] = {x=-19.084, y=-4.754, z=117.183, rx=179.992, ry=0.024, rz=-143.254, fatherId=FrmDraw[0]}
  [639] = {x=-19.205, y=-4.86, z=117.177, rx=179.99, ry=0.03, rz=-141.952, fatherId=FrmDraw[0]}
  [640] = {x=-19.331, y=-4.968, z=117.171, rx=179.987, ry=0.037, rz=-140.654, fatherId=FrmDraw[0]}
  [641] = {x=-19.454, y=-5.071, z=117.165, rx=179.983, ry=0.045, rz=-139.438, fatherId=FrmDraw[0]}
  [642] = {x=-19.597, y=-5.186, z=117.157, rx=179.979, ry=0.055, rz=-138.098, fatherId=FrmDraw[0]}
  [643] = {x=-19.731, y=-5.289, z=117.15, rx=179.974, ry=0.067, rz=-136.902, fatherId=FrmDraw[0]}
  [644] = {x=-19.878, y=-5.397, z=117.141, rx=179.967, ry=0.082, rz=-135.669, fatherId=FrmDraw[0]}
  [645] = {x=-20.046, y=-5.511, z=117.131, rx=179.957, ry=0.102, rz=-134.357, fatherId=FrmDraw[0]}
  [646] = {x=-20.191, y=-5.602, z=117.122, rx=179.947, ry=0.122, rz=-133.296, fatherId=FrmDraw[0]}
  [647] = {x=-20.367, y=-5.705, z=117.11, rx=179.934, ry=0.149, rz=-132.102, fatherId=FrmDraw[0]}
  [648] = {x=-20.519, y=-5.814, z=117.1, rx=179.921, ry=0.174, rz=-131.127, fatherId=FrmDraw[0]}
  [649] = {x=-20.699, y=-5.986, z=117.087, rx=179.904, ry=0.205, rz=-130.024, fatherId=FrmDraw[0]}
  [650] = {x=-20.858, y=-6.19, z=117.075, rx=179.889, ry=0.233, rz=-129.097, fatherId=FrmDraw[0]}
  [651] = {x=-21.001, y=-6.437, z=117.063, rx=179.875, ry=0.259, rz=-128.303, fatherId=FrmDraw[0]}
  [652] = {x=-21.119, y=-6.698, z=117.053, rx=179.862, ry=0.28, rz=-127.683, fatherId=FrmDraw[0]}
  [653] = {x=-21.234, y=-6.983, z=117.043, rx=179.85, ry=0.301, rz=-127.107, fatherId=FrmDraw[0]}
  [654] = {x=-21.33, y=-7.253, z=117.034, rx=179.84, ry=0.319, rz=-126.638, fatherId=FrmDraw[0]}
  [655] = {x=-21.434, y=-7.593, z=117.025, rx=179.829, ry=0.337, rz=-126.141, fatherId=FrmDraw[0]}
  [656] = {x=-21.511, y=-7.9, z=117.018, rx=179.821, ry=0.349, rz=-125.768, fatherId=FrmDraw[0]}
  [657] = {x=-21.578, y=-8.217, z=117.011, rx=179.816, ry=0.357, rz=-125.43, fatherId=FrmDraw[0]}
  [658] = {x=-21.658, y=-8.588, z=117.004, rx=179.81, ry=0.366, rz=-125.02, fatherId=FrmDraw[0]}
  [659] = {x=-21.732, y=-8.918, z=116.998, rx=179.805, ry=0.372, rz=-124.641, fatherId=FrmDraw[0]}
  [660] = {x=-21.801, y=-9.216, z=116.992, rx=179.801, ry=0.377, rz=-124.284, fatherId=FrmDraw[0]}
  [661] = {x=-21.876, y=-9.53, z=116.987, rx=179.797, ry=0.381, rz=-123.897, fatherId=FrmDraw[0]}
  [662] = {x=-21.882, y=-9.521, z=117.484, rx=179.795, ry=0.384, rz=-123.896, fatherId=FrmDraw[0]}
  [663] = {x=-21.888, y=-9.513, z=117.981, rx=179.794, ry=0.387, rz=-123.895, fatherId=FrmDraw[0]}
  [664] = {x=-21.893, y=-9.506, z=118.379, rx=179.792, ry=0.389, rz=-123.894, fatherId=FrmDraw[0]}
  [665] = {x=-21.898, y=-9.499, z=118.777, rx=179.791, ry=0.392, rz=-123.893, fatherId=FrmDraw[0]}
  [666] = {x=-21.901, y=-9.495, z=119.014, rx=179.79, ry=0.393, rz=-123.892, fatherId=FrmDraw[0]}
  [667] = {x=-21.906, y=-9.489, z=119.373, rx=179.789, ry=0.396, rz=-123.892, fatherId=FrmDraw[0]}
  [668] = {x=-21.912, y=-9.481, z=119.848, rx=179.788, ry=0.398, rz=-123.891, fatherId=FrmDraw[0]}
  [669] = {x=-21.918, y=-9.473, z=120.297, rx=179.786, ry=0.401, rz=-123.89, fatherId=FrmDraw[0]}
  [670] = {x=-21.923, y=-9.467, z=120.668, rx=179.785, ry=0.403, rz=-123.889, fatherId=FrmDraw[0]}
  [671] = {x=-21.928, y=-9.46, z=121.039, rx=179.784, ry=0.406, rz=-123.888, fatherId=FrmDraw[0]}
  [672] = {x=-21.845, y=-9.093, z=121.045, rx=179.788, ry=0.402, rz=-124.325, fatherId=FrmDraw[0]}
  [673] = {x=-21.769, y=-8.74, z=121.052, rx=179.792, ry=0.397, rz=-124.728, fatherId=FrmDraw[0]}
  [674] = {x=-21.697, y=-8.391, z=121.058, rx=179.797, ry=0.391, rz=-125.108, fatherId=FrmDraw[0]}
  [675] = {x=-21.638, y=-8.102, z=121.063, rx=179.802, ry=0.385, rz=-125.409, fatherId=FrmDraw[0]}
  [676] = {x=-21.575, y=-7.782, z=121.069, rx=179.807, ry=0.377, rz=-125.73, fatherId=FrmDraw[0]}
  [677] = {x=-21.509, y=-7.482, z=121.076, rx=179.813, ry=0.367, rz=-126.051, fatherId=FrmDraw[0]}
  [678] = {x=-21.413, y=-7.146, z=121.085, rx=179.824, ry=0.35, rz=-126.502, fatherId=FrmDraw[0]}
  [679] = {x=-21.303, y=-6.836, z=121.095, rx=179.836, ry=0.33, rz=-127.021, fatherId=FrmDraw[0]}
  [680] = {x=-21.191, y=-6.564, z=121.105, rx=179.848, ry=0.308, rz=-127.572, fatherId=FrmDraw[0]}
  [681] = {x=-21.071, y=-6.308, z=121.115, rx=179.861, ry=0.286, rz=-128.189, fatherId=FrmDraw[0]}
  [682] = {x=-20.932, y=-6.069, z=121.126, rx=179.875, ry=0.261, rz=-128.946, fatherId=FrmDraw[0]}
  [683] = {x=-20.773, y=-5.866, z=121.138, rx=179.891, ry=0.232, rz=-129.864, fatherId=FrmDraw[0]}
  [684] = {x=-20.59, y=-5.697, z=121.152, rx=179.909, ry=0.201, rz=-130.968, fatherId=FrmDraw[0]}
  [685] = {x=-20.419, y=-5.583, z=121.164, rx=179.924, ry=0.172, rz=-132.053, fatherId=FrmDraw[0]}
  [686] = {x=-20.23, y=-5.492, z=121.176, rx=179.939, ry=0.141, rz=-133.307, fatherId=FrmDraw[0]}
  [687] = {x=-20.054, y=-5.404, z=121.187, rx=179.952, ry=0.115, rz=-134.556, fatherId=FrmDraw[0]}
  [688] = {x=-19.877, y=-5.305, z=121.198, rx=179.963, ry=0.093, rz=-135.914, fatherId=FrmDraw[0]}
  [689] = {x=-19.712, y=-5.201, z=121.207, rx=179.971, ry=0.074, rz=-137.273, fatherId=FrmDraw[0]}
  [690] = {x=-19.569, y=-5.104, z=121.215, rx=179.977, ry=0.061, rz=-138.523, fatherId=FrmDraw[0]}
  [691] = {x=-19.444, y=-5.013, z=121.222, rx=179.982, ry=0.05, rz=-139.689, fatherId=FrmDraw[0]}
  [692] = {x=-19.298, y=-4.901, z=121.23, rx=179.986, ry=0.04, rz=-141.114, fatherId=FrmDraw[0]}
  [693] = {x=-19.179, y=-4.805, z=121.236, rx=179.989, ry=0.033, rz=-142.336, fatherId=FrmDraw[0]}
  [694] = {x=-19.074, y=-4.717, z=121.241, rx=179.991, ry=0.028, rz=-143.461, fatherId=FrmDraw[0]}
  [695] = {x=-18.958, y=-4.618, z=121.246, rx=179.993, ry=0.023, rz=-144.749, fatherId=FrmDraw[0]}
  [696] = {x=-18.847, y=-4.521, z=121.251, rx=179.994, ry=0.019, rz=-146.026, fatherId=FrmDraw[0]}
  [697] = {x=-18.726, y=-4.408, z=121.257, rx=179.995, ry=0.015, rz=-147.486, fatherId=FrmDraw[0]}
  [698] = {x=-18.617, y=-4.297, z=121.262, rx=179.996, ry=0.014, rz=-148.881, fatherId=FrmDraw[0]}
  [699] = {x=-18.518, y=-4.187, z=121.266, rx=179.996, ry=0.014, rz=-150.22, fatherId=FrmDraw[0]}
  [700] = {x=-18.428, y=-4.079, z=121.269, rx=179.996, ry=0.015, rz=-151.511, fatherId=FrmDraw[0]}
  [701] = {x=-18.346, y=-3.973, z=121.272, rx=179.996, ry=0.018, rz=-152.759, fatherId=FrmDraw[0]}
  [702] = {x=-18.25, y=-3.838, z=121.276, rx=179.995, ry=0.023, rz=-154.311, fatherId=FrmDraw[0]}
  [703] = {x=-18.184, y=-3.736, z=121.278, rx=179.994, ry=0.029, rz=-155.473, fatherId=FrmDraw[0]}
  [704] = {x=-18.124, y=-3.635, z=121.28, rx=179.993, ry=0.035, rz=-156.607, fatherId=FrmDraw[0]}
  [705] = {x=-18.07, y=-3.536, z=121.281, rx=179.992, ry=0.042, rz=-157.716, fatherId=FrmDraw[0]}
  [706] = {x=-17.998, y=-3.393, z=121.282, rx=179.99, ry=0.054, rz=-159.311, fatherId=FrmDraw[0]}
  [707] = {x=-17.935, y=-3.25, z=121.283, rx=179.989, ry=0.068, rz=-160.916, fatherId=FrmDraw[0]}
  [708] = {x=-17.88, y=-3.116, z=121.283, rx=179.987, ry=0.083, rz=-162.465, fatherId=FrmDraw[0]}
  [709] = {x=-17.832, y=-2.989, z=121.283, rx=179.986, ry=0.099, rz=-163.999, fatherId=FrmDraw[0]}
  [710] = {x=-17.789, y=-2.868, z=121.283, rx=179.985, ry=0.116, rz=-165.512, fatherId=FrmDraw[0]}
  [711] = {x=-17.752, y=-2.754, z=121.282, rx=179.985, ry=0.134, rz=-167.01, fatherId=FrmDraw[0]}
  [712] = {x=-17.72, y=-2.646, z=121.28, rx=179.985, ry=0.152, rz=-168.496, fatherId=FrmDraw[0]}
  [713] = {x=-17.692, y=-2.545, z=121.279, rx=179.985, ry=0.171, rz=-169.972, fatherId=FrmDraw[0]}
  [714] = {x=-17.668, y=-2.449, z=121.277, rx=179.986, ry=0.19, rz=-171.441, fatherId=FrmDraw[0]}
  [715] = {x=-17.648, y=-2.36, z=121.275, rx=179.987, ry=0.21, rz=-172.903, fatherId=FrmDraw[0]}
  [716] = {x=-17.631, y=-2.277, z=121.272, rx=179.989, ry=0.23, rz=-174.36, fatherId=FrmDraw[0]}
  [717] = {x=-17.618, y=-2.198, z=121.269, rx=179.991, ry=0.251, rz=-175.808, fatherId=FrmDraw[0]}
  [718] = {x=-17.612, y=-2.118, z=121.266, rx=179.993, ry=0.274, rz=-177.225, fatherId=FrmDraw[0]}
  [719] = {x=-17.612, y=-2.038, z=121.262, rx=179.996, ry=0.298, rz=-178.614, fatherId=FrmDraw[0]}
  [720] = {x=-17.621, y=-1.93, z=121.257, rx=-179.999, ry=0.331, rz=179.575, fatherId=FrmDraw[0]}
  [721] = {x=-17.638, y=-1.823, z=121.25, rx=-179.993, ry=0.367, rz=177.803, fatherId=FrmDraw[0]}
  [722] = {x=-17.664, y=-1.717, z=121.244, rx=-179.986, ry=0.404, rz=176.064, fatherId=FrmDraw[0]}
  [723] = {x=-17.695, y=-1.613, z=121.236, rx=-179.978, ry=0.442, rz=174.351, fatherId=FrmDraw[0]}
  [724] = {x=-17.729, y=-1.512, z=121.229, rx=-179.969, ry=0.479, rz=172.658, fatherId=FrmDraw[0]}
  [725] = {x=-17.763, y=-1.413, z=121.222, rx=-179.959, ry=0.514, rz=170.982, fatherId=FrmDraw[0]}
  [726] = {x=-17.796, y=-1.317, z=121.215, rx=-179.949, ry=0.547, rz=169.318, fatherId=FrmDraw[0]}
  [727] = {x=-17.826, y=-1.22, z=121.209, rx=-179.938, ry=0.577, rz=167.683, fatherId=FrmDraw[0]}
  [728] = {x=-17.857, y=-1.115, z=121.203, rx=-179.926, ry=0.605, rz=166.103, fatherId=FrmDraw[0]}
  [729] = {x=-17.891, y=-1.003, z=121.197, rx=-179.914, ry=0.632, rz=164.577, fatherId=FrmDraw[0]}
  [730] = {x=-17.927, y=-0.883, z=121.191, rx=-179.902, ry=0.658, rz=163.102, fatherId=FrmDraw[0]}
  [731] = {x=-17.966, y=-0.756, z=121.185, rx=-179.89, ry=0.684, rz=161.676, fatherId=FrmDraw[0]}
  [732] = {x=-18.01, y=-0.622, z=121.179, rx=-179.877, ry=0.71, rz=160.296, fatherId=FrmDraw[0]}
  [733] = {x=-18.058, y=-0.482, z=121.172, rx=-179.863, ry=0.736, rz=158.96, fatherId=FrmDraw[0]}
  [734] = {x=-18.112, y=-0.336, z=121.166, rx=-179.85, ry=0.762, rz=157.664, fatherId=FrmDraw[0]}
  [735] = {x=-18.171, y=-0.184, z=121.159, rx=-179.835, ry=0.789, rz=156.408, fatherId=FrmDraw[0]}
  [736] = {x=-18.236, y=-0.028, z=121.152, rx=-179.82, ry=0.817, rz=155.188, fatherId=FrmDraw[0]}
  [737] = {x=-18.306, y=0.13, z=121.144, rx=-179.805, ry=0.846, rz=153.987, fatherId=FrmDraw[0]}
  [738] = {x=-18.381, y=0.285, z=121.137, rx=-179.788, ry=0.875, rz=152.777, fatherId=FrmDraw[0]}
  [739] = {x=-18.458, y=0.435, z=121.129, rx=-179.771, ry=0.903, rz=151.558, fatherId=FrmDraw[0]}
  [740] = {x=-18.54, y=0.581, z=121.121, rx=-179.753, ry=0.932, rz=150.327, fatherId=FrmDraw[0]}
  [741] = {x=-18.624, y=0.723, z=121.114, rx=-179.735, ry=0.959, rz=149.084, fatherId=FrmDraw[0]}
  [742] = {x=-18.712, y=0.86, z=121.106, rx=-179.715, ry=0.987, rz=147.828, fatherId=FrmDraw[0]}
  [743] = {x=-18.803, y=0.992, z=121.098, rx=-179.695, ry=1.014, rz=146.557, fatherId=FrmDraw[0]}
  [744] = {x=-18.898, y=1.119, z=121.09, rx=-179.675, ry=1.04, rz=145.269, fatherId=FrmDraw[0]}
  [745] = {x=-18.995, y=1.242, z=121.082, rx=-179.653, ry=1.066, rz=143.964, fatherId=FrmDraw[0]}
  [746] = {x=-19.096, y=1.359, z=121.074, rx=-179.631, ry=1.091, rz=142.641, fatherId=FrmDraw[0]}
  [747] = {x=-19.201, y=1.474, z=121.066, rx=-179.608, ry=1.116, rz=141.314, fatherId=FrmDraw[0]}
  [748] = {x=-19.311, y=1.597, z=121.057, rx=-179.584, ry=1.143, rz=140.029, fatherId=FrmDraw[0]}
  [749] = {x=-19.426, y=1.728, z=121.048, rx=-179.56, ry=1.171, rz=138.787, fatherId=FrmDraw[0]}
  [750] = {x=-19.515, y=1.831, z=121.041, rx=-179.541, ry=1.193, rz=137.884, fatherId=FrmDraw[0]}
  [751] = {x=-19.636, y=1.977, z=121.032, rx=-179.515, ry=1.222, rz=136.718, fatherId=FrmDraw[0]}
  [752] = {x=-19.76, y=2.132, z=121.023, rx=-179.489, ry=1.252, rz=135.595, fatherId=FrmDraw[0]}
  [753] = {x=-19.886, y=2.297, z=121.013, rx=-179.463, ry=1.282, rz=134.516, fatherId=FrmDraw[0]}
  [754] = {x=-20.012, y=2.472, z=121.004, rx=-179.436, ry=1.312, rz=133.48, fatherId=FrmDraw[0]}
  [755] = {x=-20.139, y=2.659, z=120.995, rx=-179.41, ry=1.341, rz=132.487, fatherId=FrmDraw[0]}
  [756] = {x=-20.266, y=2.856, z=120.986, rx=-179.384, ry=1.369, rz=131.536, fatherId=FrmDraw[0]}
  [757] = {x=-20.384, y=3.053, z=120.978, rx=-179.36, ry=1.394, rz=130.664, fatherId=FrmDraw[0]}
  [758] = {x=-20.507, y=3.265, z=120.97, rx=-179.335, ry=1.418, rz=129.754, fatherId=FrmDraw[0]}
  [759] = {x=-20.629, y=3.481, z=120.963, rx=-179.311, ry=1.44, rz=128.848, fatherId=FrmDraw[0]}
  [760] = {x=-20.75, y=3.7, z=120.956, rx=-179.287, ry=1.46, rz=127.946, fatherId=FrmDraw[0]}
  [761] = {x=-20.872, y=3.924, z=120.95, rx=-179.264, ry=1.478, rz=127.048, fatherId=FrmDraw[0]}
  [762] = {x=-20.996, y=4.15, z=120.944, rx=-179.241, ry=1.495, rz=126.155, fatherId=FrmDraw[0]}
  [763] = {x=-21.122, y=4.379, z=120.938, rx=-179.217, ry=1.512, rz=125.265, fatherId=FrmDraw[0]}
  [764] = {x=-21.251, y=4.611, z=120.932, rx=-179.194, ry=1.528, rz=124.379, fatherId=FrmDraw[0]}
  [765] = {x=-21.384, y=4.845, z=120.926, rx=-179.17, ry=1.544, rz=123.496, fatherId=FrmDraw[0]}
  [766] = {x=-21.523, y=5.081, z=120.92, rx=-179.146, ry=1.56, rz=122.619, fatherId=FrmDraw[0]}
  [767] = {x=-21.664, y=5.325, z=120.914, rx=-179.121, ry=1.579, rz=121.783, fatherId=FrmDraw[0]}
  [768] = {x=-21.804, y=5.576, z=120.908, rx=-179.096, ry=1.598, rz=121.012, fatherId=FrmDraw[0]}
  [769] = {x=-21.925, y=5.801, z=120.902, rx=-179.074, ry=1.616, rz=120.389, fatherId=FrmDraw[0]}
  [770] = {x=-22.025, y=5.996, z=120.898, rx=-179.056, ry=1.632, rz=119.897, fatherId=FrmDraw[0]}
  [771] = {x=-22.164, y=6.281, z=120.892, rx=-179.03, ry=1.654, rz=119.251, fatherId=FrmDraw[0]}
  [772] = {x=-22.281, y=6.538, z=120.887, rx=-179.009, ry=1.674, rz=118.737, fatherId=FrmDraw[0]}
  [773] = {x=-22.383, y=6.779, z=120.883, rx=-178.99, ry=1.691, rz=118.306, fatherId=FrmDraw[0]}
  [774] = {x=-22.481, y=7.031, z=120.879, rx=-178.972, ry=1.708, rz=117.907, fatherId=FrmDraw[0]}
  [775] = {x=-22.565, y=7.263, z=120.876, rx=-178.957, ry=1.722, rz=117.578, fatherId=FrmDraw[0]}
  [776] = {x=-22.664, y=7.566, z=120.873, rx=-178.938, ry=1.739, rz=117.202, fatherId=FrmDraw[0]}
  [777] = {x=-22.739, y=7.817, z=120.871, rx=-178.925, ry=1.752, rz=116.922, fatherId=FrmDraw[0]}
  [778] = {x=-22.828, y=8.137, z=120.869, rx=-178.909, ry=1.765, rz=116.585, fatherId=FrmDraw[0]}
  [779] = {x=-22.896, y=8.399, z=120.868, rx=-178.898, ry=1.775, rz=116.326, fatherId=FrmDraw[0]}
  [780] = {x=-22.977, y=8.733, z=120.867, rx=-178.885, ry=1.785, rz=116.016, fatherId=FrmDraw[0]}
  [781] = {x=-23.04, y=9.006, z=120.866, rx=-178.875, ry=1.793, rz=115.779, fatherId=FrmDraw[0]}
  [782] = {x=-23.114, y=9.353, z=120.866, rx=-178.863, ry=1.801, rz=115.496, fatherId=FrmDraw[0]}
  [783] = {x=-23.172, y=9.636, z=120.867, rx=-178.855, ry=1.807, rz=115.281, fatherId=FrmDraw[0]}
  [784] = {x=-23.241, y=9.995, z=120.867, rx=-178.845, ry=1.814, rz=115.026, fatherId=FrmDraw[0]}
  [785] = {x=-23.295, y=10.287, z=120.868, rx=-178.837, ry=1.82, rz=114.833, fatherId=FrmDraw[0]}
  [786] = {x=-23.36, y=10.657, z=120.868, rx=-178.827, ry=1.827, rz=114.607, fatherId=FrmDraw[0]}
  [787] = {x=-23.411, y=10.956, z=120.869, rx=-178.82, ry=1.832, rz=114.438, fatherId=FrmDraw[0]}
  [788] = {x=-23.475, y=11.334, z=120.87, rx=-178.811, ry=1.84, rz=114.235, fatherId=FrmDraw[0]}
  [789] = {x=-23.528, y=11.637, z=120.871, rx=-178.803, ry=1.846, rz=114.071, fatherId=FrmDraw[0]}
  [790] = {x=-23.595, y=12.015, z=120.873, rx=-178.793, ry=1.853, rz=113.864, fatherId=FrmDraw[0]}
  [791] = {x=-23.657, y=12.356, z=120.874, rx=-178.785, ry=1.859, rz=113.675, fatherId=FrmDraw[0]}
  [792] = {x=-23.72, y=12.697, z=120.875, rx=-178.776, ry=1.866, rz=113.485, fatherId=FrmDraw[0]}
  [793] = {x=-23.785, y=13.039, z=120.876, rx=-178.768, ry=1.872, rz=113.292, fatherId=FrmDraw[0]}
  [794] = {x=-23.852, y=13.381, z=120.878, rx=-178.759, ry=1.878, rz=113.098, fatherId=FrmDraw[0]}
  [795] = {x=-23.92, y=13.723, z=120.879, rx=-178.751, ry=1.884, rz=112.902, fatherId=FrmDraw[0]}
  [796] = {x=-23.989, y=14.066, z=120.88, rx=-178.742, ry=1.89, rz=112.703, fatherId=FrmDraw[0]}
  [797] = {x=-24.06, y=14.41, z=120.882, rx=-178.734, ry=1.895, rz=112.503, fatherId=FrmDraw[0]}
  [798] = {x=-24.132, y=14.754, z=120.884, rx=-178.725, ry=1.901, rz=112.3, fatherId=FrmDraw[0]}
  [799] = {x=-24.205, y=15.098, z=120.885, rx=-178.717, ry=1.906, rz=112.095, fatherId=FrmDraw[0]}
  [800] = {x=-24.28, y=15.443, z=120.887, rx=-178.709, ry=1.91, rz=111.888, fatherId=FrmDraw[0]}
  [801] = {x=-24.357, y=15.789, z=120.889, rx=-178.701, ry=1.915, rz=111.679, fatherId=FrmDraw[0]}
  [802] = {x=-24.434, y=16.135, z=120.891, rx=-178.693, ry=1.919, rz=111.468, fatherId=FrmDraw[0]}
  [803] = {x=-24.504, y=16.444, z=120.893, rx=-178.686, ry=1.922, rz=111.278, fatherId=FrmDraw[0]}
  [804] = {x=-24.593, y=16.831, z=120.895, rx=-178.677, ry=1.926, rz=111.038, fatherId=FrmDraw[0]}
  [805] = {x=-24.666, y=17.141, z=120.897, rx=-178.671, ry=1.929, rz=110.844, fatherId=FrmDraw[0]}
  [806] = {x=-24.758, y=17.529, z=120.899, rx=-178.663, ry=1.931, rz=110.599, fatherId=FrmDraw[0]}
  [807] = {x=-24.833, y=17.841, z=120.901, rx=-178.656, ry=1.933, rz=110.401, fatherId=FrmDraw[0]}
  [808] = {x=-24.928, y=18.232, z=120.904, rx=-178.649, ry=1.935, rz=110.151, fatherId=FrmDraw[0]}
  [809] = {x=-25.004, y=18.546, z=120.906, rx=-178.643, ry=1.936, rz=109.95, fatherId=FrmDraw[0]}
  [810] = {x=-25.099, y=18.941, z=120.909, rx=-178.636, ry=1.937, rz=109.702, fatherId=FrmDraw[0]}
  [811] = {x=-25.175, y=19.259, z=120.911, rx=-178.631, ry=1.938, rz=109.507, fatherId=FrmDraw[0]}
  [812] = {x=-25.27, y=19.66, z=120.914, rx=-178.624, ry=1.938, rz=109.268, fatherId=FrmDraw[0]}
  [813] = {x=-25.347, y=19.982, z=120.917, rx=-178.619, ry=1.939, rz=109.079, fatherId=FrmDraw[0]}
  [814] = {x=-25.442, y=20.388, z=120.92, rx=-178.612, ry=1.94, rz=108.847, fatherId=FrmDraw[0]}
  [815] = {x=-25.519, y=20.713, z=120.923, rx=-178.607, ry=1.941, rz=108.665, fatherId=FrmDraw[0]}
  [816] = {x=-25.616, y=21.122, z=120.926, rx=-178.599, ry=1.943, rz=108.442, fatherId=FrmDraw[0]}
  [817] = {x=-25.695, y=21.451, z=120.928, rx=-178.593, ry=1.945, rz=108.267, fatherId=FrmDraw[0]}
  [818] = {x=-25.795, y=21.863, z=120.932, rx=-178.585, ry=1.949, rz=108.052, fatherId=FrmDraw[0]}
  [819] = {x=-25.876, y=22.194, z=120.934, rx=-178.578, ry=1.953, rz=107.883, fatherId=FrmDraw[0]}
  [820] = {x=-25.98, y=22.607, z=120.938, rx=-178.569, ry=1.957, rz=107.673, fatherId=FrmDraw[0]}
  [821] = {x=-26.063, y=22.939, z=120.941, rx=-178.562, ry=1.961, rz=107.505, fatherId=FrmDraw[0]}
  [822] = {x=-26.167, y=23.357, z=120.944, rx=-178.553, ry=1.966, rz=107.296, fatherId=FrmDraw[0]}
  [823] = {x=-26.266, y=23.765, z=120.948, rx=-178.546, ry=1.968, rz=107.095, fatherId=FrmDraw[0]}
  [824] = {x=-26.349, y=24.12, z=120.951, rx=-178.541, ry=1.969, rz=106.922, fatherId=FrmDraw[0]}
  [825] = {x=-26.44, y=24.538, z=120.955, rx=-178.537, ry=1.967, rz=106.722, fatherId=FrmDraw[0]}
  [826] = {x=-26.514, y=24.903, z=120.959, rx=-178.536, ry=1.962, rz=106.55, fatherId=FrmDraw[0]}
  [827] = {x=-26.587, y=25.305, z=120.963, rx=-178.537, ry=1.954, rz=106.365, fatherId=FrmDraw[0]}
  [828] = {x=-26.667, y=25.705, z=120.967, rx=-178.542, ry=1.94, rz=106.15, fatherId=FrmDraw[0]}
  [829] = {x=-26.663, y=25.706, z=121.384, rx=-178.542, ry=1.941, rz=106.158, fatherId=FrmDraw[0]}
  [830] = {x=-26.659, y=25.708, z=121.801, rx=-178.542, ry=1.941, rz=106.166, fatherId=FrmDraw[0]}
  [831] = {x=-26.656, y=25.71, z=122.168, rx=-178.542, ry=1.941, rz=106.174, fatherId=FrmDraw[0]}
  [832] = {x=-26.652, y=25.711, z=122.585, rx=-178.542, ry=1.941, rz=106.182, fatherId=FrmDraw[0]}
  [833] = {x=-26.649, y=25.713, z=122.951, rx=-178.542, ry=1.941, rz=106.189, fatherId=FrmDraw[0]}
  [834] = {x=-26.645, y=25.714, z=123.369, rx=-178.542, ry=1.941, rz=106.198, fatherId=FrmDraw[0]}
  [835] = {x=-26.64, y=25.716, z=123.843, rx=-178.542, ry=1.941, rz=106.207, fatherId=FrmDraw[0]}
  [836] = {x=-26.636, y=25.718, z=124.292, rx=-178.543, ry=1.942, rz=106.216, fatherId=FrmDraw[0]}
  [837] = {x=-26.633, y=25.719, z=124.657, rx=-178.543, ry=1.942, rz=106.223, fatherId=FrmDraw[0]}
  [838] = {x=-26.629, y=25.721, z=125.023, rx=-178.543, ry=1.942, rz=106.231, fatherId=FrmDraw[0]}
  [839] = {x=-26.566, y=25.344, z=125.019, rx=-178.537, ry=1.956, rz=106.418, fatherId=FrmDraw[0]}
  [840] = {x=-26.51, y=24.896, z=125.015, rx=-178.534, ry=1.966, rz=106.575, fatherId=FrmDraw[0]}
  [841] = {x=-26.451, y=24.52, z=125.011, rx=-178.534, ry=1.97, rz=106.716, fatherId=FrmDraw[0]}
  [842] = {x=-26.372, y=24.093, z=125.006, rx=-178.538, ry=1.972, rz=106.887, fatherId=FrmDraw[0]}
  [843] = {x=-26.297, y=23.732, z=125.003, rx=-178.543, ry=1.971, rz=107.04, fatherId=FrmDraw[0]}
  [844] = {x=-26.203, y=23.321, z=124.999, rx=-178.55, ry=1.967, rz=107.225, fatherId=FrmDraw[0]}
  [845] = {x=-26.101, y=22.902, z=124.995, rx=-178.56, ry=1.962, rz=107.424, fatherId=FrmDraw[0]}
  [846] = {x=-26.016, y=22.57, z=124.992, rx=-178.567, ry=1.957, rz=107.588, fatherId=FrmDraw[0]}
  [847] = {x=-25.909, y=22.159, z=124.989, rx=-178.577, ry=1.951, rz=107.802, fatherId=FrmDraw[0]}
  [848] = {x=-25.824, y=21.831, z=124.987, rx=-178.585, ry=1.947, rz=107.977, fatherId=FrmDraw[0]}
  [849] = {x=-25.72, y=21.422, z=124.983, rx=-178.593, ry=1.944, rz=108.201, fatherId=FrmDraw[0]}
  [850] = {x=-25.639, y=21.096, z=124.981, rx=-178.599, ry=1.942, rz=108.382, fatherId=FrmDraw[0]}
  [851] = {x=-25.539, y=20.688, z=124.978, rx=-178.606, ry=1.94, rz=108.611, fatherId=FrmDraw[0]}
  [852] = {x=-25.462, y=20.363, z=124.975, rx=-178.611, ry=1.939, rz=108.796, fatherId=FrmDraw[0]}
  [853] = {x=-25.366, y=19.958, z=124.972, rx=-178.618, ry=1.939, rz=109.03, fatherId=FrmDraw[0]}
  [854] = {x=-25.29, y=19.635, z=124.969, rx=-178.623, ry=1.939, rz=109.22, fatherId=FrmDraw[0]}
  [855] = {x=-25.196, y=19.234, z=124.966, rx=-178.629, ry=1.939, rz=109.459, fatherId=FrmDraw[0]}
  [856] = {x=-25.122, y=18.914, z=124.964, rx=-178.634, ry=1.938, rz=109.652, fatherId=FrmDraw[0]}
  [857] = {x=-25.028, y=18.518, z=124.961, rx=-178.64, ry=1.938, rz=109.896, fatherId=FrmDraw[0]}
  [858] = {x=-24.953, y=18.202, z=124.959, rx=-178.646, ry=1.937, rz=110.093, fatherId=FrmDraw[0]}
  [859] = {x=-24.86, y=17.81, z=124.956, rx=-178.653, ry=1.936, rz=110.338, fatherId=FrmDraw[0]}
  [860] = {x=-24.787, y=17.497, z=124.954, rx=-178.659, ry=1.934, rz=110.533, fatherId=FrmDraw[0]}
  [861] = {x=-24.696, y=17.107, z=124.951, rx=-178.667, ry=1.931, rz=110.773, fatherId=FrmDraw[0]}
  [862] = {x=-24.624, y=16.796, z=124.949, rx=-178.674, ry=1.928, rz=110.963, fatherId=FrmDraw[0]}
  [863] = {x=-24.535, y=16.409, z=124.947, rx=-178.682, ry=1.924, rz=111.199, fatherId=FrmDraw[0]}
  [864] = {x=-24.465, y=16.1, z=124.945, rx=-178.689, ry=1.921, rz=111.386, fatherId=FrmDraw[0]}
  [865] = {x=-24.379, y=15.714, z=124.943, rx=-178.698, ry=1.916, rz=111.617, fatherId=FrmDraw[0]}
  [866] = {x=-24.311, y=15.407, z=124.941, rx=-178.706, ry=1.912, rz=111.8, fatherId=FrmDraw[0]}
  [867] = {x=-24.228, y=15.023, z=124.939, rx=-178.715, ry=1.906, rz=112.027, fatherId=FrmDraw[0]}
  [868] = {x=-24.162, y=14.717, z=124.938, rx=-178.723, ry=1.901, rz=112.207, fatherId=FrmDraw[0]}
  [869] = {x=-24.081, y=14.335, z=124.936, rx=-178.732, ry=1.895, rz=112.43, fatherId=FrmDraw[0]}
  [870] = {x=-24.018, y=14.03, z=124.935, rx=-178.74, ry=1.89, rz=112.606, fatherId=FrmDraw[0]}
  [871] = {x=-23.94, y=13.649, z=124.933, rx=-178.749, ry=1.883, rz=112.825, fatherId=FrmDraw[0]}
  [872] = {x=-23.879, y=13.345, z=124.932, rx=-178.757, ry=1.878, rz=112.998, fatherId=FrmDraw[0]}
  [873] = {x=-23.804, y=12.965, z=124.93, rx=-178.767, ry=1.871, rz=113.213, fatherId=FrmDraw[0]}
  [874] = {x=-23.746, y=12.662, z=124.929, rx=-178.775, ry=1.865, rz=113.383, fatherId=FrmDraw[0]}
  [875] = {x=-23.674, y=12.283, z=124.928, rx=-178.784, ry=1.858, rz=113.594, fatherId=FrmDraw[0]}
  [876] = {x=-23.618, y=11.98, z=124.927, rx=-178.792, ry=1.852, rz=113.761, fatherId=FrmDraw[0]}
  [877] = {x=-23.55, y=11.602, z=124.926, rx=-178.802, ry=1.844, rz=113.969, fatherId=FrmDraw[0]}
  [878] = {x=-23.497, y=11.3, z=124.925, rx=-178.809, ry=1.838, rz=114.133, fatherId=FrmDraw[0]}
  [879] = {x=-23.433, y=10.923, z=124.924, rx=-178.818, ry=1.831, rz=114.337, fatherId=FrmDraw[0]}
  [880] = {x=-23.381, y=10.623, z=124.923, rx=-178.826, ry=1.826, rz=114.507, fatherId=FrmDraw[0]}
  [881] = {x=-23.315, y=10.253, z=124.922, rx=-178.835, ry=1.819, rz=114.731, fatherId=FrmDraw[0]}
  [882] = {x=-23.262, y=9.96, z=124.921, rx=-178.843, ry=1.813, rz=114.92, fatherId=FrmDraw[0]}
  [883] = {x=-23.193, y=9.599, z=124.921, rx=-178.853, ry=1.806, rz=115.168, fatherId=FrmDraw[0]}
  [884] = {x=-23.136, y=9.315, z=124.921, rx=-178.861, ry=1.8, rz=115.376, fatherId=FrmDraw[0]}
  [885] = {x=-23.063, y=8.965, z=124.921, rx=-178.873, ry=1.792, rz=115.648, fatherId=FrmDraw[0]}
  [886] = {x=-23.002, y=8.689, z=124.921, rx=-178.883, ry=1.784, rz=115.874, fatherId=FrmDraw[0]}
  [887] = {x=-22.922, y=8.351, z=124.922, rx=-178.896, ry=1.773, rz=116.168, fatherId=FrmDraw[0]}
  [888] = {x=-22.855, y=8.085, z=124.923, rx=-178.907, ry=1.763, rz=116.411, fatherId=FrmDraw[0]}
  [889] = {x=-22.767, y=7.76, z=124.925, rx=-178.923, ry=1.749, rz=116.727, fatherId=FrmDraw[0]}
  [890] = {x=-22.693, y=7.505, z=124.927, rx=-178.936, ry=1.736, rz=116.989, fatherId=FrmDraw[0]}
  [891] = {x=-22.595, y=7.198, z=124.93, rx=-178.954, ry=1.718, rz=117.348, fatherId=FrmDraw[0]}
  [892] = {x=-22.511, y=6.963, z=124.933, rx=-178.97, ry=1.703, rz=117.665, fatherId=FrmDraw[0]}
  [893] = {x=-22.401, y=6.681, z=124.937, rx=-178.99, ry=1.685, rz=118.1, fatherId=FrmDraw[0]}
  [894] = {x=-22.268, y=6.37, z=124.943, rx=-179.014, ry=1.662, rz=118.66, fatherId=FrmDraw[0]}
  [895] = {x=-22.169, y=6.158, z=124.947, rx=-179.032, ry=1.646, rz=119.094, fatherId=FrmDraw[0]}
  [896] = {x=-22.049, y=5.914, z=124.952, rx=-179.054, ry=1.627, rz=119.652, fatherId=FrmDraw[0]}
  [897] = {x=-21.908, y=5.644, z=124.958, rx=-179.079, ry=1.606, rz=120.352, fatherId=FrmDraw[0]}
  [898] = {x=-21.763, y=5.382, z=124.964, rx=-179.105, ry=1.586, rz=121.122, fatherId=FrmDraw[0]}
  [899] = {x=-21.619, y=5.133, z=124.971, rx=-179.13, ry=1.567, rz=121.949, fatherId=FrmDraw[0]}
  [900] = {x=-21.477, y=4.896, z=124.977, rx=-179.155, ry=1.55, rz=122.824, fatherId=FrmDraw[0]}
  [901] = {x=-21.34, y=4.662, z=124.983, rx=-179.179, ry=1.534, rz=123.711, fatherId=FrmDraw[0]}
  [902] = {x=-21.208, y=4.43, z=124.988, rx=-179.203, ry=1.518, rz=124.596, fatherId=FrmDraw[0]}
  [903] = {x=-21.078, y=4.199, z=124.994, rx=-179.226, ry=1.502, rz=125.482, fatherId=FrmDraw[0]}
  [904] = {x=-20.952, y=3.971, z=125.001, rx=-179.25, ry=1.485, rz=126.368, fatherId=FrmDraw[0]}
  [905] = {x=-20.827, y=3.745, z=125.007, rx=-179.273, ry=1.466, rz=127.255, fatherId=FrmDraw[0]}
  [906] = {x=-20.703, y=3.521, z=125.014, rx=-179.297, ry=1.446, rz=128.142, fatherId=FrmDraw[0]}
  [907] = {x=-20.58, y=3.301, z=125.021, rx=-179.321, ry=1.424, rz=129.03, fatherId=FrmDraw[0]}
  [908] = {x=-20.455, y=3.084, z=125.029, rx=-179.346, ry=1.4, rz=129.92, fatherId=FrmDraw[0]}
  [909] = {x=-20.329, y=2.87, z=125.037, rx=-179.371, ry=1.374, rz=130.811, fatherId=FrmDraw[0]}
  [910] = {x=-20.208, y=2.676, z=125.045, rx=-179.396, ry=1.347, rz=131.684, fatherId=FrmDraw[0]}
  [911] = {x=-20.08, y=2.483, z=125.054, rx=-179.422, ry=1.318, rz=132.648, fatherId=FrmDraw[0]}
  [912] = {x=-19.952, y=2.301, z=125.064, rx=-179.448, ry=1.289, rz=133.658, fatherId=FrmDraw[0]}
  [913] = {x=-19.824, y=2.131, z=125.073, rx=-179.475, ry=1.259, rz=134.714, fatherId=FrmDraw[0]}
  [914] = {x=-19.699, y=1.972, z=125.082, rx=-179.501, ry=1.23, rz=135.817, fatherId=FrmDraw[0]}
  [915] = {x=-19.576, y=1.822, z=125.092, rx=-179.527, ry=1.2, rz=136.966, fatherId=FrmDraw[0]}
  [916] = {x=-19.457, y=1.682, z=125.101, rx=-179.552, ry=1.172, rz=138.161, fatherId=FrmDraw[0]}
  [917] = {x=-19.399, y=1.616, z=125.105, rx=-179.564, ry=1.158, rz=138.777, fatherId=FrmDraw[0]}
  [918] = {x=-19.285, y=1.49, z=125.114, rx=-179.589, ry=1.131, rz=140.042, fatherId=FrmDraw[0]}
  [919] = {x=-19.176, y=1.373, z=125.122, rx=-179.612, ry=1.106, rz=141.353, fatherId=FrmDraw[0]}
  [920] = {x=-19.072, y=1.259, z=125.13, rx=-179.635, ry=1.081, rz=142.688, fatherId=FrmDraw[0]}
  [921] = {x=-18.971, y=1.141, z=125.138, rx=-179.657, ry=1.055, rz=144.005, fatherId=FrmDraw[0]}
  [922] = {x=-18.872, y=1.018, z=125.146, rx=-179.679, ry=1.029, rz=145.304, fatherId=FrmDraw[0]}
  [923] = {x=-18.777, y=0.889, z=125.154, rx=-179.699, ry=1.002, rz=146.586, fatherId=FrmDraw[0]}
  [924] = {x=-18.684, y=0.756, z=125.163, rx=-179.719, ry=0.974, rz=147.852, fatherId=FrmDraw[0]}
  [925] = {x=-18.595, y=0.619, z=125.17, rx=-179.739, ry=0.946, rz=149.104, fatherId=FrmDraw[0]}
  [926] = {x=-18.51, y=0.477, z=125.178, rx=-179.757, ry=0.918, rz=150.343, fatherId=FrmDraw[0]}
  [927] = {x=-18.427, y=0.33, z=125.186, rx=-179.775, ry=0.889, rz=151.571, fatherId=FrmDraw[0]}
  [928] = {x=-18.349, y=0.18, z=125.194, rx=-179.792, ry=0.861, rz=152.788, fatherId=FrmDraw[0]}
  [929] = {x=-18.275, y=0.026, z=125.201, rx=-179.808, ry=0.832, rz=153.997, fatherId=FrmDraw[0]}
  [930] = {x=-18.205, y=-0.131, z=125.209, rx=-179.823, ry=0.803, rz=155.207, fatherId=FrmDraw[0]}
  [931] = {x=-18.142, y=-0.284, z=125.216, rx=-179.838, ry=0.776, rz=156.448, fatherId=FrmDraw[0]}
  [932] = {x=-18.086, y=-0.432, z=125.222, rx=-179.852, ry=0.75, rz=157.723, fatherId=FrmDraw[0]}
  [933] = {x=-18.034, y=-0.574, z=125.229, rx=-179.866, ry=0.724, rz=159.035, fatherId=FrmDraw[0]}
  [934] = {x=-17.987, y=-0.712, z=125.235, rx=-179.879, ry=0.699, rz=160.385, fatherId=FrmDraw[0]}
  [935] = {x=-17.945, y=-0.843, z=125.241, rx=-179.892, ry=0.674, rz=161.777, fatherId=FrmDraw[0]}
  [936] = {x=-17.906, y=-0.968, z=125.247, rx=-179.904, ry=0.648, rz=163.212, fatherId=FrmDraw[0]}
  [937] = {x=-17.869, y=-1.087, z=125.253, rx=-179.917, ry=0.621, rz=164.692, fatherId=FrmDraw[0]}
  [938] = {x=-17.834, y=-1.199, z=125.259, rx=-179.928, ry=0.593, rz=166.221, fatherId=FrmDraw[0]}
  [939] = {x=-17.8, y=-1.304, z=125.266, rx=-179.94, ry=0.564, rz=167.801, fatherId=FrmDraw[0]}
  [940] = {x=-17.765, y=-1.404, z=125.272, rx=-179.951, ry=0.532, rz=169.423, fatherId=FrmDraw[0]}
  [941] = {x=-17.727, y=-1.504, z=125.28, rx=-179.961, ry=0.497, rz=171.067, fatherId=FrmDraw[0]}
  [942] = {x=-17.69, y=-1.605, z=125.287, rx=-179.971, ry=0.46, rz=172.733, fatherId=FrmDraw[0]}
  [943] = {x=-17.655, y=-1.707, z=125.295, rx=-179.979, ry=0.422, rz=174.427, fatherId=FrmDraw[0]}
  [944] = {x=-17.625, y=-1.809, z=125.302, rx=-179.987, ry=0.385, rz=176.153, fatherId=FrmDraw[0]}
  [945] = {x=-17.604, y=-1.911, z=125.308, rx=-179.994, ry=0.349, rz=177.913, fatherId=FrmDraw[0]}
  [946] = {x=-17.591, y=-2.014, z=125.314, rx=-179.999, ry=0.315, rz=179.71, fatherId=FrmDraw[0]}
  [947] = {x=-17.588, y=-2.116, z=125.319, rx=179.996, ry=0.284, rz=-178.451, fatherId=FrmDraw[0]}
  [948] = {x=-17.593, y=-2.192, z=125.322, rx=179.993, ry=0.261, rz=-177.039, fatherId=FrmDraw[0]}
  [949] = {x=-17.604, y=-2.267, z=125.325, rx=179.991, ry=0.241, rz=-175.597, fatherId=FrmDraw[0]}
  [950] = {x=-17.619, y=-2.345, z=125.328, rx=179.989, ry=0.221, rz=-174.138, fatherId=FrmDraw[0]}
  [951] = {x=-17.638, y=-2.428, z=125.33, rx=179.987, ry=0.201, rz=-172.675, fatherId=FrmDraw[0]}
  [952] = {x=-17.66, y=-2.517, z=125.332, rx=179.986, ry=0.182, rz=-171.208, fatherId=FrmDraw[0]}
  [953] = {x=-17.686, y=-2.612, z=125.334, rx=179.985, ry=0.163, rz=-169.733, fatherId=FrmDraw[0]}
  [954] = {x=-17.716, y=-2.713, z=125.335, rx=179.985, ry=0.145, rz=-168.25, fatherId=FrmDraw[0]}
  [955] = {x=-17.75, y=-2.82, z=125.336, rx=179.985, ry=0.127, rz=-166.757, fatherId=FrmDraw[0]}
  [956] = {x=-17.789, y=-2.934, z=125.337, rx=179.986, ry=0.11, rz=-165.25, fatherId=FrmDraw[0]}
  [957] = {x=-17.833, y=-3.054, z=125.338, rx=179.987, ry=0.093, rz=-163.727, fatherId=FrmDraw[0]}
  [958] = {x=-17.883, y=-3.181, z=125.338, rx=179.988, ry=0.078, rz=-162.184, fatherId=FrmDraw[0]}
  [959] = {x=-17.94, y=-3.312, z=125.337, rx=179.989, ry=0.063, rz=-160.636, fatherId=FrmDraw[0]}
  [960] = {x=-18.006, y=-3.452, z=125.337, rx=179.991, ry=0.05, rz=-159.018, fatherId=FrmDraw[0]}
  [961] = {x=-18.081, y=-3.589, z=125.335, rx=179.992, ry=0.038, rz=-157.421, fatherId=FrmDraw[0]}
  [962] = {x=-18.137, y=-3.685, z=125.333, rx=179.993, ry=0.032, rz=-156.307, fatherId=FrmDraw[0]}
  [963] = {x=-18.199, y=-3.782, z=125.332, rx=179.994, ry=0.026, rz=-155.167, fatherId=FrmDraw[0]}
  [964] = {x=-18.267, y=-3.88, z=125.329, rx=179.995, ry=0.022, rz=-153.999, fatherId=FrmDraw[0]}
  [965] = {x=-18.365, y=-4.01, z=125.326, rx=179.996, ry=0.017, rz=-152.435, fatherId=FrmDraw[0]}
  [966] = {x=-18.45, y=-4.112, z=125.323, rx=179.996, ry=0.015, rz=-151.181, fatherId=FrmDraw[0]}
  [967] = {x=-18.542, y=-4.216, z=125.319, rx=179.996, ry=0.014, rz=-149.885, fatherId=FrmDraw[0]}
  [968] = {x=-18.643, y=-4.321, z=125.315, rx=179.996, ry=0.014, rz=-148.54, fatherId=FrmDraw[0]}
  [969] = {x=-18.755, y=-4.427, z=125.31, rx=179.995, ry=0.016, rz=-147.139, fatherId=FrmDraw[0]}
  [970] = {x=-18.878, y=-4.535, z=125.304, rx=179.994, ry=0.02, rz=-145.674, fatherId=FrmDraw[0]}
  [971] = {x=-19.01, y=-4.645, z=125.298, rx=179.992, ry=0.025, rz=-144.177, fatherId=FrmDraw[0]}
  [972] = {x=-19.107, y=-4.723, z=125.294, rx=179.99, ry=0.03, rz=-143.115, fatherId=FrmDraw[0]}
  [973] = {x=-19.218, y=-4.808, z=125.288, rx=179.987, ry=0.036, rz=-141.964, fatherId=FrmDraw[0]}
  [974] = {x=-19.354, y=-4.908, z=125.281, rx=179.984, ry=0.046, rz=-140.605, fatherId=FrmDraw[0]}
  [975] = {x=-19.499, y=-5.005, z=125.273, rx=179.979, ry=0.058, rz=-139.248, fatherId=FrmDraw[0]}
  [976] = {x=-19.654, y=-5.101, z=125.265, rx=179.972, ry=0.073, rz=-137.874, fatherId=FrmDraw[0]}
  [977] = {x=-19.807, y=-5.186, z=125.256, rx=179.964, ry=0.09, rz=-136.608, fatherId=FrmDraw[0]}
  [978] = {x=-19.967, y=-5.265, z=125.247, rx=179.955, ry=0.11, rz=-135.363, fatherId=FrmDraw[0]}
  [979] = {x=-20.149, y=-5.343, z=125.235, rx=179.942, ry=0.136, rz=-134.032, fatherId=FrmDraw[0]}
  [980] = {x=-20.364, y=-5.424, z=125.222, rx=179.925, ry=0.17, rz=-132.579, fatherId=FrmDraw[0]}
  [981] = {x=-20.532, y=-5.511, z=125.21, rx=179.911, ry=0.198, rz=-131.491, fatherId=FrmDraw[0]}
  [982] = {x=-20.715, y=-5.648, z=125.197, rx=179.894, ry=0.229, rz=-130.351, fatherId=FrmDraw[0]}
  [983] = {x=-20.882, y=-5.823, z=125.185, rx=179.878, ry=0.258, rz=-129.365, fatherId=FrmDraw[0]}
  [984] = {x=-21.03, y=-6.037, z=125.173, rx=179.863, ry=0.285, rz=-128.524, fatherId=FrmDraw[0]}
  [985] = {x=-21.152, y=-6.267, z=125.163, rx=179.85, ry=0.307, rz=-127.874, fatherId=FrmDraw[0]}
  [986] = {x=-21.267, y=-6.517, z=125.153, rx=179.837, ry=0.328, rz=-127.293, fatherId=FrmDraw[0]}
  [987] = {x=-21.382, y=-6.815, z=125.143, rx=179.825, ry=0.35, rz=-126.739, fatherId=FrmDraw[0]}
  [988] = {x=-21.48, y=-7.132, z=125.134, rx=179.814, ry=0.367, rz=-126.276, fatherId=FrmDraw[0]}
  [989] = {x=-21.543, y=-7.396, z=125.128, rx=179.807, ry=0.378, rz=-125.972, fatherId=FrmDraw[0]}
  [990] = {x=-21.598, y=-7.692, z=125.122, rx=179.802, ry=0.385, rz=-125.695, fatherId=FrmDraw[0]}
  [991] = {x=-21.665, y=-8.058, z=125.116, rx=179.797, ry=0.393, rz=-125.347, fatherId=FrmDraw[0]}
  [992] = {x=-21.733, y=-8.421, z=125.109, rx=179.792, ry=0.399, rz=-124.984, fatherId=FrmDraw[0]}
  [993] = {x=-21.787, y=-8.696, z=125.105, rx=179.789, ry=0.403, rz=-124.695, fatherId=FrmDraw[0]}
  [994] = {x=-21.858, y=-9.046, z=125.099, rx=179.785, ry=0.407, rz=-124.311, fatherId=FrmDraw[0]}
  [995] = {x=-21.936, y=-9.408, z=125.093, rx=179.782, ry=0.41, rz=-123.894, fatherId=FrmDraw[0]}
  [996] = {x=-21.933, y=-9.407, z=125.51, rx=179.782, ry=0.408, rz=-123.892, fatherId=FrmDraw[0]}
  [997] = {x=-21.93, y=-9.405, z=125.928, rx=179.783, ry=0.407, rz=-123.891, fatherId=FrmDraw[0]}
  [998] = {x=-21.927, y=-9.404, z=126.295, rx=179.784, ry=0.405, rz=-123.89, fatherId=FrmDraw[0]}
  [999] = {x=-21.924, y=-9.403, z=126.712, rx=179.785, ry=0.404, rz=-123.888, fatherId=FrmDraw[0]}
  [1000] = {x=-21.921, y=-9.402, z=127.079, rx=179.785, ry=0.403, rz=-123.887, fatherId=FrmDraw[0]}
  [1001] = {x=-21.918, y=-9.401, z=127.497, rx=179.786, ry=0.401, rz=-123.886, fatherId=FrmDraw[0]}
  [1002] = {x=-21.914, y=-9.399, z=127.97, rx=179.787, ry=0.399, rz=-123.884, fatherId=FrmDraw[0]}
  [1003] = {x=-21.911, y=-9.398, z=128.42, rx=179.788, ry=0.398, rz=-123.882, fatherId=FrmDraw[0]}
  [1004] = {x=-21.908, y=-9.397, z=128.785, rx=179.789, ry=0.396, rz=-123.881, fatherId=FrmDraw[0]}
  [1005] = {x=-21.905, y=-9.396, z=129.151, rx=179.789, ry=0.395, rz=-123.88, fatherId=FrmDraw[0]}
  [1006] = {x=-21.841, y=-9.094, z=129.156, rx=179.792, ry=0.392, rz=-124.222, fatherId=FrmDraw[0]}
  [1007] = {x=-21.767, y=-8.722, z=129.162, rx=179.796, ry=0.389, rz=-124.623, fatherId=FrmDraw[0]}
  [1008] = {x=-21.698, y=-8.35, z=129.168, rx=179.8, ry=0.384, rz=-125.001, fatherId=FrmDraw[0]}
  [1009] = {x=-21.636, y=-7.996, z=129.174, rx=179.804, ry=0.379, rz=-125.341, fatherId=FrmDraw[0]}
  [1010] = {x=-21.574, y=-7.627, z=129.18, rx=179.808, ry=0.373, rz=-125.674, fatherId=FrmDraw[0]}
  [1011] = {x=-21.527, y=-7.331, z=129.186, rx=179.812, ry=0.368, rz=-125.928, fatherId=FrmDraw[0]}
  [1012] = {x=-21.474, y=-7.055, z=129.191, rx=179.817, ry=0.36, rz=-126.199, fatherId=FrmDraw[0]}
  [1013] = {x=-21.387, y=-6.733, z=129.199, rx=179.826, ry=0.346, rz=-126.623, fatherId=FrmDraw[0]}
